  MoveL 3945 to (-46.24, -29.98, -6) mm, rotated rx -180 ry 0 rz 90 deg; joints [72.382, -18.215, 87.048, 0, 21.167, 72.382]
  MoveL 3946 to (-46.24, -29.98, -3) mm, rotated rx 180 ry 0 rz 90 deg; joints [72.382, -18.371, 87.15, 0, 21.221, 72.382]
  Establecer velocidad (1000.0 mm/s)
  MoveL 3947 to (-46.24, -29.98, 10) mm, rotated rx -180 ry 0 rz 90 deg; joints [72.382, -19.042, 87.583, 0, 21.46, 72.382]
  Establecer velocidad (66.7 mm/s)
  MoveL 3948 to (17.19, -67.01, 10) mm, rotated rx 180 ry 0 rz 90 deg; joints [71.851, -17.649, 82.287, 0, 25.361, 71.851]
  MoveL 3949 to (17.19, -67.01, -2.75) mm, rotated rx -180 ry 0 rz 90 deg; joints [71.851, -17.004, 81.861, 0, 25.143, 71.851]
  MoveL 3950 to (17.02, -68.52, -3.16) mm, rotated rx 180 ry 0 rz 90 deg; joints [71.803, -16.977, 81.823, 0, 25.153, 71.803]
  MoveL 3951 to (17.22, -70.03, -3.56) mm, rotated rx 180 ry 0 rz 90 deg; joints [71.757, -16.942, 81.759, 0, 25.183, 71.757]
  MoveL 3952 to (17.75, -71.45, -3.97) mm, rotated rx -180 ry 0 rz 90 deg; joints [71.718, -16.902, 81.673, 0, 25.228, 71.718]
  MoveL 3953 to (18.58, -72.72, -4.37) mm, rotated rx 180 ry 0 rz 90 deg; joints [71.687, -16.856, 81.569, 0, 25.287, 71.687]
  MoveL 3954 to (19.67, -73.78, -4.78) mm, rotated rx 180 ry 0 rz 90 deg; joints [71.665, -16.806, 81.451, 0, 25.356, 71.665]
  MoveL 3955 to (20.97, -74.57, -5.19) mm, rotated rx 180 ry 0 rz 90 deg; joints [71.654, -16.754, 81.324, 0, 25.431, 71.654]
  MoveL 3956 to (22.42, -75.05, -5.59) mm, rotated rx -180 ry 0 rz 90 deg; joints [71.654, -16.701, 81.194, 0, 25.508, 71.654]
  MoveL 3957 to (23.93, -75.17, -6) mm, rotated rx -180 ry 0 rz 90 deg; joints [71.666, -16.649, 81.067, 0, 25.582, 71.666]
  MoveL 3958 to (43.12, -74.95, -6) mm, rotated rx -180 ry 0 rz 90 deg; joints [71.869, -16.251, 79.664, 0, 26.587, 71.869]
  MoveL 3959 to (50.7, -74.82, -6) mm, rotated rx 180 ry 0 rz 90 deg; joints [71.949, -16.089, 79.105, 0, 26.984, 71.949]
  MoveC 3960 to (53.51, -71.7, -6) mm, rotated rx 180 ry 0 rz 90 deg; joints [72.073, -16.05, 78.971, 0, 27.079, 72.073] to (53.65, -67.5, -6) mm, rotated rx 180 ry 0 rz 90 deg; joints [72.203, -16.076, 79.061, 0, 27.015, 72.203]
  MoveL 3961 to (53.54, -67.37, -6) mm, rotated rx -180 ry 0 rz 90 deg; joints [72.206, -16.08, 79.072, 0, 27.007, 72.206]
  MoveL 3962 to (28.6, -38.38, -6) mm, rotated rx -180 ry 0 rz 90 deg; joints [72.864, -16.793, 81.584, 0, 25.21, 72.864]
  MoveL 3963 to (26.1, -35.54, -6) mm, rotated rx 180 ry 0 rz 90 deg; joints [72.929, -16.861, 81.829, 0, 25.032, 72.929]
  MoveL 3964 to (11.85, -24.12, -6) mm, rotated rx 180 ry 0 rz 90 deg; joints [73.154, -17.209, 83.109, 0, 24.1, 73.154]
  MoveC 3965 to (10.01, -23.4, -6) mm, rotated rx 180 ry 0 rz 90 deg; joints [73.159, -17.248, 83.256, 0, 23.993, 73.159] to (8.05, -23.61, -6) mm, rotated rx 180 ry 0 rz 90 deg; joints [73.133, -17.284, 83.391, 0, 23.893, 73.133]
  MoveL 3966 to (7.26, -23.95, -6) mm, rotated rx 180 ry 0 rz 90 deg; joints [73.115, -17.297, 83.44, 0, 23.857, 73.115]
  MoveC 3967 to (6.07, -24.83, -6) mm, rotated rx 180 ry 0 rz 90 deg; joints [73.075, -17.315, 83.507, 0, 23.808, 73.075] to (5.36, -26.14, -6) mm, rotated rx -180 ry 0 rz 90 deg; joints [73.026, -17.321, 83.528, 0, 23.792, 73.026]
  MoveL 3968 to (5.21, -26.67, -6) mm, rotated rx -180 ry 0 rz 90 deg; joints [73.008, -17.321, 83.528, 0, 23.793, 73.008]
  MoveL 3969 to (-6.22, -69.65, -6) mm, rotated rx -180 ry 0 rz 90 deg; joints [71.524, -17.277, 83.363, 0, 23.914, 71.524]
  MoveL 3970 to (-6.48, -70.6, -6) mm, rotated rx 180 ry 0 rz 90 deg; joints [71.492, -17.276, 83.359, 0, 23.917, 71.492]
  MoveC 3971 to (-5.7, -73.8, -6) mm, rotated rx -180 ry 0 rz 90 deg; joints [71.399, -17.241, 83.227, 0, 24.013, 71.399] to (-2.85, -75.47, -6) mm, rotated rx 180 ry 0 rz 90 deg; joints [71.376, -17.176, 82.985, 0, 24.19, 71.376]
  MoveL 3972 to (-2.37, -75.48, -6) mm, rotated rx 180 ry 0 rz 90 deg; joints [71.381, -17.167, 82.951, 0, 24.215, 71.381]
  MoveL 3973 to (23.93, -75.17, -6) mm, rotated rx -180 ry 0 rz 90 deg; joints [71.666, -16.649, 81.067, 0, 25.582, 71.666]
  MoveL 3974 to (23.84, -67.62, -6) mm, rotated rx -180 ry 0 rz 90 deg; joints [71.9, -16.702, 81.254, 0, 25.447, 71.9]
  MoveL 3975 to (23.84, -67.62, -3) mm, rotated rx 180 ry 0 rz 90 deg; joints [71.9, -16.853, 81.356, 0, 25.497, 71.9]
  Establecer velocidad (1000.0 mm/s)
  MoveL 3976 to (23.84, -67.62, 10) mm, rotated rx 180 ry 0 rz 90 deg; joints [71.9, -17.51, 81.791, 0, 25.718, 71.9]
  Establecer velocidad (66.7 mm/s)
  MoveL 3977 to (65.32, -31.32, 10) mm, rotated rx -180 ry 0 rz 90 deg; joints [73.432, -16.868, 79.565, 0, 27.303, 73.432]
  MoveL 3978 to (65.32, -31.32, -2.75) mm, rotated rx 180 ry 0 rz 90 deg; joints [73.432, -16.229, 79.136, 0, 27.093, 73.432]
  MoveL 3979 to (66.82, -31.5, -3.16) mm, rotated rx -180 ry 0 rz 90 deg; joints [73.44, -16.174, 79.005, 0, 27.17, 73.44]
  MoveL 3980 to (68.33, -31.32, -3.56) mm, rotated rx -180 ry 0 rz 90 deg; joints [73.459, -16.122, 78.881, 0, 27.24, 73.459]
  MoveL 3981 to (69.76, -30.81, -3.97) mm, rotated rx 180 ry 0 rz 90 deg; joints [73.488, -16.073, 78.771, 0, 27.302, 73.488]
  MoveL 3982 to (71.04, -29.99, -4.37) mm, rotated rx 180 ry 0 rz 90 deg; joints [73.525, -16.03, 78.679, 0, 27.351, 73.525]
  MoveL 3983 to (72.11, -28.92, -4.78) mm, rotated rx 180 ry 0 rz 90 deg; joints [73.568, -15.993, 78.608, 0, 27.385, 73.568]
  MoveL 3984 to (72.92, -27.63, -5.19) mm, rotated rx 180 ry 0 rz 90 deg; joints [73.615, -15.963, 78.562, 0, 27.401, 73.615]
  MoveL 3985 to (73.42, -26.19, -5.59) mm, rotated rx -180 ry 0 rz 90 deg; joints [73.664, -15.941, 78.542, 0, 27.399, 73.664]
  MoveL 3986 to (73.56, -24.68, -6) mm, rotated rx -180 ry 0 rz 90 deg; joints [73.712, -15.927, 78.551, 0, 27.376, 73.712]
  MoveL 3987 to (73.56, -10.28, -6) mm, rotated rx 180 ry 0 rz 90 deg; joints [74.158, -16.019, 78.865, 0, 27.154, 74.158]
  MoveC 3988 to (71.61, -7.6, -6) mm, rotated rx -180 ry 0 rz 90 deg; joints [74.224, -16.079, 79.069, 0, 27.01, 74.224] to (68.7, -6.02, -6) mm, rotated rx 180 ry 0 rz 90 deg; joints [74.248, -16.152, 79.322, 0, 26.83, 74.248]
  MoveC 3989 to (67.33, -5.86, -6) mm, rotated rx 180 ry 0 rz 90 deg; joints [74.241, -16.183, 79.429, 0, 26.754, 74.241] to (65.97, -6.14, -6) mm, rotated rx 180 ry 0 rz 90 deg; joints [74.22, -16.211, 79.525, 0, 26.686, 74.22]
  MoveL 3990 to (64.91, -7.57, -6) mm, rotated rx -180 ry 0 rz 90 deg; joints [74.166, -16.225, 79.574, 0, 26.651, 74.166]
  MoveL 3991 to (54.87, -21.32, -6) mm, rotated rx -180 ry 0 rz 90 deg; joints [73.646, -16.355, 80.028, 0, 26.327, 73.646]
  MoveL 3992 to (53.21, -23.57, -6) mm, rotated rx -180 ry 0 rz 90 deg; joints [73.561, -16.376, 80.102, 0, 26.275, 73.561]
  MoveC 3993 to (52.43, -26.14, -6) mm, rotated rx 180 ry 0 rz 90 deg; joints [73.474, -16.377, 80.103, 0, 26.274, 73.474] to (53.45, -28.63, -6) mm, rotated rx 180 ry 0 rz 90 deg; joints [73.406, -16.34, 79.973, 0, 26.367, 73.406]
  MoveL 3994 to (66.39, -43.19, -6) mm, rotated rx 180 ry 0 rz 90 deg; joints [73.075, -15.964, 78.676, 0, 27.288, 73.075]
  MoveC 3995 to (68.56, -43.36, -6) mm, rotated rx 180 ry 0 rz 90 deg; joints [73.09, -15.915, 78.508, 0, 27.407, 73.09] to (70.6, -42.58, -6) mm, rotated rx 180 ry 0 rz 90 deg; joints [73.133, -15.875, 78.372, 0, 27.503, 73.133]
  MoveL 3996 to (71.01, -42.29, -6) mm, rotated rx -180 ry 0 rz 90 deg; joints [73.146, -15.867, 78.348, 0, 27.52, 73.146]
  MoveC 3997 to (72.52, -40.87, -6) mm, rotated rx 180 ry 0 rz 90 deg; joints [73.203, -15.843, 78.266, 0, 27.577, 73.203] to (73.56, -39.08, -6) mm, rotated rx -180 ry 0 rz 90 deg; joints [73.268, -15.832, 78.228, 0, 27.604, 73.268]
  MoveL 3998 to (73.56, -24.68, -6) mm, rotated rx -180 ry 0 rz 90 deg; joints [73.712, -15.927, 78.551, 0, 27.376, 73.712]
  MoveL 3999 to (66.01, -24.68, -6) mm, rotated rx 180 ry 0 rz 90 deg; joints [73.644, -16.094, 79.121, 0, 26.973, 73.644]
  MoveL 4000 to (66.01, -24.68, -3) mm, rotated rx 180 ry 0 rz 90 deg; joints [73.644, -16.244, 79.223, 0, 27.021, 73.644]
  Establecer velocidad (1000.0 mm/s)
  MoveL 4001 to (66.01, -24.68, 10) mm, rotated rx -180 ry 0 rz 90 deg; joints [73.644, -16.896, 79.66, 0, 27.236, 73.644]
  Establecer velocidad (66.7 mm/s)
  MoveL 4002 to (37.19, 22.66, 10) mm, rotated rx 180 ry 0 rz 90 deg; joints [74.878, -17.786, 82.781, 0, 25.005, 74.878]
  MoveL 4003 to (37.19, 22.66, -2.75) mm, rotated rx -180 ry 0 rz 90 deg; joints [74.878, -17.14, 82.354, 0, 24.785, 74.878]
  MoveL 4004 to (37.34, 24.17, -3.16) mm, rotated rx -180 ry 0 rz 90 deg; joints [74.928, -17.124, 82.36, 0, 24.765, 74.928]
  MoveL 4005 to (37.12, 25.67, -3.56) mm, rotated rx 180 ry 0 rz 90 deg; joints [74.974, -17.116, 82.391, 0, 24.725, 74.974]
  MoveL 4006 to (36.57, 27.09, -3.97) mm, rotated rx -180 ry 0 rz 90 deg; joints [75.015, -17.114, 82.445, 0, 24.669, 75.015]
  MoveL 4007 to (35.73, 28.35, -4.37) mm, rotated rx 180 ry 0 rz 90 deg; joints [75.048, -17.117, 82.518, 0, 24.599, 75.048]
  MoveL 4008 to (34.62, 29.4, -4.78) mm, rotated rx 180 ry 0 rz 90 deg; joints [75.072, -17.124, 82.605, 0, 24.519, 75.072]
  MoveL 4009 to (33.31, 30.17, -5.19) mm, rotated rx -180 ry 0 rz 90 deg; joints [75.085, -17.133, 82.701, 0, 24.432, 75.085]
  MoveL 4010 to (31.87, 30.63, -5.59) mm, rotated rx 180 ry 0 rz 90 deg; joints [75.088, -17.143, 82.802, 0, 24.342, 75.088]
  MoveL 4011 to (30.35, 30.74, -6) mm, rotated rx 180 ry 0 rz 90 deg; joints [75.078, -17.153, 82.9, 0, 24.253, 75.078]
  MoveL 4012 to (9, 30.22, -6) mm, rotated rx 180 ry 0 rz 90 deg; joints [74.876, -17.556, 84.425, 0, 23.131, 74.876]
  MoveC 4013 to (5.64, 28.68, -6) mm, rotated rx 180 ry 0 rz 90 deg; joints [74.797, -17.611, 84.634, 0, 22.976, 74.797] to (4.7, 25.11, -6) mm, rotated rx 180 ry 0 rz 90 deg; joints [74.672, -17.61, 84.632, 0, 22.978, 74.672]
  MoveL 4014 to (5.03, 24.17, -6) mm, rotated rx -180 ry 0 rz 90 deg; joints [74.645, -17.599, 84.59, 0, 23.009, 74.645]
  MoveL 4015 to (10.58, 8.87, -6) mm, rotated rx 180 ry 0 rz 90 deg; joints [74.2, -17.417, 83.891, 0, 23.526, 74.2]
  MoveC 4016 to (11.12, 7.86, -6) mm, rotated rx 180 ry 0 rz 90 deg; joints [74.172, -17.401, 83.832, 0, 23.569, 74.172] to (11.92, 7.03, -6) mm, rotated rx 180 ry 0 rz 90 deg; joints [74.153, -17.382, 83.758, 0, 23.624, 74.153]
  MoveL 4017 to (28.28, -5.64, -6) mm, rotated rx 180 ry 0 rz 90 deg; joints [73.897, -16.995, 82.317, 0, 24.678, 73.897]
  MoveC 4018 to (30.24, -6.45, -6) mm, rotated rx -180 ry 0 rz 90 deg; joints [73.889, -16.951, 82.158, 0, 24.794, 73.889] to (32.34, -6.16, -6) mm, rotated rx -180 ry 0 rz 90 deg; joints [73.918, -16.911, 82.011, 0, 24.9, 73.918]
  MoveC 4019 to (33.47, -5.59, -6) mm, rotated rx 180 ry 0 rz 90 deg; joints [73.946, -16.892, 81.941, 0, 24.951, 73.946] to (34.36, -4.69, -6) mm, rotated rx 180 ry 0 rz 90 deg; joints [73.983, -16.879, 81.895, 0, 24.984, 73.983]
  MoveL 4020 to (54.3, 23.22, -6) mm, rotated rx -180 ry 0 rz 90 deg; joints [75.042, -16.63, 80.997, 0, 25.633, 75.042]
  MoveL 4021 to (54.77, 23.88, -6) mm, rotated rx 180 ry 0 rz 90 deg; joints [75.067, -16.624, 80.975, 0, 25.648, 75.067]
  MoveC 4022 to (55.09, 24.53, -6) mm, rotated rx 180 ry 0 rz 90 deg; joints [75.09, -16.621, 80.964, 0, 25.656, 75.09] to (55.2, 25.24, -6) mm, rotated rx 180 ry 0 rz 90 deg; joints [75.114, -16.622, 80.97, 0, 25.652, 75.114]
  MoveL 4023 to (55.21, 25.78, -6) mm, rotated rx 180 ry 0 rz 90 deg; joints [75.131, -16.625, 80.98, 0, 25.645, 75.131]
  MoveC 4024 to (54.27, 29.03, -6) mm, rotated rx 180 ry 0 rz 90 deg; joints [75.226, -16.662, 81.113, 0, 25.549, 75.226] to (51.7, 31.24, -6) mm, rotated rx -180 ry 0 rz 90 deg; joints [75.275, -16.727, 81.346, 0, 25.381, 75.275]
  MoveL 4025 to (49.75, 31.21, -6) mm, rotated rx 180 ry 0 rz 90 deg; joints [75.258, -16.767, 81.49, 0, 25.277, 75.258]
  MoveL 4026 to (30.35, 30.74, -6) mm, rotated rx 180 ry 0 rz 90 deg; joints [75.078, -17.153, 82.9, 0, 24.253, 75.078]
  MoveL 4027 to (30.54, 23.19, -6) mm, rotated rx 180 ry 0 rz 90 deg; joints [74.838, -17.109, 82.739, 0, 24.37, 74.838]
  MoveL 4028 to (30.54, 23.19, -3) mm, rotated rx 180 ry 0 rz 90 deg; joints [74.838, -17.262, 82.841, 0, 24.421, 74.838]
  Establecer velocidad (1000.0 mm/s)
  MoveL 4029 to (30.54, 23.19, 10) mm, rotated rx 180 ry 0 rz 90 deg; joints [74.838, -17.922, 83.275, 0, 24.647, 74.838]
  Establecer velocidad (66.7 mm/s)
  MoveL 4030 to (26.5, 66.74, 10) mm, rotated rx 180 ry 0 rz 90 deg; joints [76.21, -18.22, 84.38, 0, 23.84, 76.21]
  MoveL 4031 to (26.5, 66.74, -2.75) mm, rotated rx 180 ry 0 rz 90 deg; joints [76.21, -17.57, 83.955, 0, 23.615, 76.21]
  MoveL 4032 to (26.71, 68.24, -3.16) mm, rotated rx 180 ry 0 rz 90 deg; joints [76.261, -17.553, 83.953, 0, 23.6, 76.261]
  MoveL 4033 to (26.54, 69.75, -3.56) mm, rotated rx 180 ry 0 rz 90 deg; joints [76.309, -17.542, 83.978, 0, 23.564, 76.309]
  MoveL 4034 to (26.05, 71.19, -3.97) mm, rotated rx -180 ry 0 rz 90 deg; joints [76.352, -17.537, 84.025, 0, 23.513, 76.352]
  MoveL 4035 to (25.25, 72.48, -4.37) mm, rotated rx 180 ry 0 rz 90 deg; joints [76.387, -17.538, 84.092, 0, 23.446, 76.387]
  MoveL 4036 to (24.18, 73.57, -4.78) mm, rotated rx 180 ry 0 rz 90 deg; joints [76.414, -17.542, 84.173, 0, 23.369, 76.414]
  MoveL 4037 to (22.9, 74.39, -5.19) mm, rotated rx -180 ry 0 rz 90 deg; joints [76.431, -17.549, 84.266, 0, 23.283, 76.431]
  MoveL 4038 to (21.47, 74.9, -5.59) mm, rotated rx -180 ry 0 rz 90 deg; joints [76.437, -17.558, 84.364, 0, 23.194, 76.437]
  MoveL 4039 to (19.96, 75.06, -6) mm, rotated rx -180 ry 0 rz 90 deg; joints [76.43, -17.566, 84.461, 0, 23.105, 76.43]
  MoveL 4040 to (12.79, 75.15, -6) mm, rotated rx 180 ry 0 rz 90 deg; joints [76.376, -17.698, 84.976, 0, 22.723, 76.376]
  MoveL 4041 to (-28.9, 75.59, -6) mm, rotated rx -180 ry 0 rz 90 deg; joints [76.051, -18.421, 87.908, 0, 20.513, 76.051]
  MoveL 4042 to (-29.63, 75.59, -6) mm, rotated rx -180 ry 0 rz 90 deg; joints [76.045, -18.433, 87.958, 0, 20.475, 76.045]
  MoveC 4043 to (-32.33, 72.16, -6) mm, rotated rx 180 ry 0 rz 90 deg; joints [75.907, -18.463, 88.086, 0, 20.377, 75.907] to (-31.86, 67.82, -6) mm, rotated rx -180 ry 0 rz 90 deg; joints [75.765, -18.438, 87.978, 0, 20.46, 75.765]
  MoveL 4044 to (-10.84, 54.49, -6) mm, rotated rx 180 ry 0 rz 90 deg; joints [75.5, -18.027, 86.281, 0, 21.747, 75.5]
  MoveC 4045 to (-9.04, 53.75, -6) mm, rotated rx 180 ry 0 rz 90 deg; joints [75.491, -17.993, 86.141, 0, 21.852, 75.491] to (-7.11, 53.59, -6) mm, rotated rx -180 ry 0 rz 90 deg; joints [75.502, -17.958, 86.002, 0, 21.956, 75.502]
  MoveL 4046 to (37.91, 56.91, -6) mm, rotated rx -180 ry 0 rz 90 deg; joints [75.984, -17.137, 82.841, 0, 24.296, 75.984]
  MoveC 4047 to (53.8, 58.26, -6) mm, rotated rx -180 ry 0 rz 90 deg; joints [76.153, -16.825, 81.7, 0, 25.126, 76.153] to (69.65, 59.95, -6) mm, rotated rx -180 ry 0 rz 90 deg; joints [76.331, -16.504, 80.551, 0, 25.953, 76.331]
  MoveC 4048 to (71.89, 61.11, -6) mm, rotated rx -180 ry 0 rz 90 deg; joints [76.385, -16.463, 80.405, 0, 26.058, 76.385] to (72.78, 63.46, -6) mm, rotated rx 180 ry 0 rz 90 deg; joints [76.467, -16.456, 80.38, 0, 26.075, 76.467]
  MoveL 4049 to (72.78, 69.65, -6) mm, rotated rx 180 ry 0 rz 90 deg; joints [76.663, -16.487, 80.491, 0, 25.996, 76.663]
  MoveL 4050 to (72.76, 70.26, -6) mm, rotated rx -180 ry 0 rz 90 deg; joints [76.682, -16.491, 80.503, 0, 25.987, 76.682]
  MoveC 4051 to (71.8, 72.55, -6) mm, rotated rx 180 ry 0 rz 90 deg; joints [76.748, -16.523, 80.617, 0, 25.906, 76.748] to (69.53, 73.57, -6) mm, rotated rx -180 ry 0 rz 90 deg; joints [76.763, -16.575, 80.804, 0, 25.771, 76.763]
  MoveC 4052 to (45.44, 74.54, -6) mm, rotated rx 180 ry 0 rz 90 deg; joints [76.612, -17.073, 82.605, 0, 24.468, 76.612] to (21.32, 75.04, -6) mm, rotated rx -180 ry 0 rz 90 deg; joints [76.44, -17.54, 84.363, 0, 23.177, 76.44]
  MoveL 4053 to (19.96, 75.06, -6) mm, rotated rx -180 ry 0 rz 90 deg; joints [76.43, -17.566, 84.461, 0, 23.105, 76.43]
  MoveL 4054 to (19.87, 67.51, -6) mm, rotated rx -180 ry 0 rz 90 deg; joints [76.182, -17.533, 84.336, 0, 23.197, 76.182]
  MoveL 4055 to (19.87, 67.51, -3) mm, rotated rx 180 ry 0 rz 90 deg; joints [76.182, -17.687, 84.437, 0, 23.249, 76.182]
  Establecer velocidad (1000.0 mm/s)
  MoveL 4056 to (19.87, 67.51, 10) mm, rotated rx 180 ry 0 rz 90 deg; joints [76.182, -18.351, 84.871, 0, 23.48, 76.182]
  Establecer velocidad (66.7 mm/s)
  MoveL 4057 to (26.49, 66.5, 10) mm, rotated rx -180 ry 0 rz 90 deg; joints [76.203, -18.219, 84.377, 0, 23.843, 76.203]
  MoveL 4058 to (26.49, 66.5, -3) mm, rotated rx 180 ry 0 rz 90 deg; joints [76.203, -17.557, 83.943, 0, 23.614, 76.203]
  MoveL 4059 to (26.7, 68, -3.41) mm, rotated rx -180 ry 0 rz 90 deg; joints [76.253, -17.539, 83.941, 0, 23.598, 76.253]
  MoveL 4060 to (26.54, 69.51, -3.81) mm, rotated rx -180 ry 0 rz 90 deg; joints [76.301, -17.528, 83.966, 0, 23.563, 76.301]
  MoveL 4061 to (26.04, 70.95, -4.22) mm, rotated rx 180 ry 0 rz 90 deg; joints [76.344, -17.524, 84.013, 0, 23.511, 76.344]
  MoveL 4062 to (25.24, 72.25, -4.63) mm, rotated rx -180 ry 0 rz 90 deg; joints [76.38, -17.524, 84.079, 0, 23.445, 76.38]
  MoveL 4063 to (24.18, 73.33, -5.03) mm, rotated rx -180 ry 0 rz 90 deg; joints [76.407, -17.528, 84.161, 0, 23.367, 76.407]
  MoveL 4064 to (22.9, 74.15, -5.44) mm, rotated rx 180 ry 0 rz 90 deg; joints [76.423, -17.535, 84.254, 0, 23.282, 76.423]
  MoveL 4065 to (21.47, 74.67, -5.84) mm, rotated rx 180 ry 0 rz 90 deg; joints [76.429, -17.544, 84.352, 0, 23.192, 76.429]
  MoveL 4066 to (19.96, 74.83, -6.25) mm, rotated rx -180 ry 0 rz 90 deg; joints [76.422, -17.552, 84.449, 0, 23.103, 76.422]
  MoveL 4067 to (16.58, 74.87, -6.25) mm, rotated rx 180 ry 0 rz 90 deg; joints [76.397, -17.615, 84.692, 0, 22.923, 76.397]
  MoveL 4068 to (-29.04, 75.36, -6.25) mm, rotated rx -180 ry 0 rz 90 deg; joints [76.042, -18.41, 87.905, 0, 20.504, 76.042]
  MoveC 4069 to (-31.69, 71.97, -6.25) mm, rotated rx -180 ry 0 rz 90 deg; joints [75.906, -18.439, 88.029, 0, 20.409, 75.906] to (-31.22, 67.7, -6.25) mm, rotated rx 180 ry 0 rz 90 deg; joints [75.766, -18.414, 87.923, 0, 20.49, 75.766]
  MoveL 4070 to (-10.9, 54.79, -6.25) mm, rotated rx 180 ry 0 rz 90 deg; joints [75.509, -18.017, 86.282, 0, 21.735, 75.509]
  MoveC 4071 to (-9.09, 53.98, -6.25) mm, rotated rx -180 ry 0 rz 90 deg; joints [75.498, -17.982, 86.14, 0, 21.842, 75.498] to (-7.11, 53.8, -6.25) mm, rotated rx -180 ry 0 rz 90 deg; joints [75.509, -17.946, 85.998, 0, 21.949, 75.509]
  MoveL 4072 to (36.88, 57.07, -6.25) mm, rotated rx 180 ry 0 rz 90 deg; joints [75.98, -17.145, 82.911, 0, 24.235, 75.98]
  MoveC 4073 to (53.18, 58.48, -6.25) mm, rotated rx -180 ry 0 rz 90 deg; joints [76.156, -16.826, 81.741, 0, 25.085, 76.156] to (69.44, 60.27, -6.25) mm, rotated rx 180 ry 0 rz 90 deg; joints [76.34, -16.498, 80.564, 0, 25.933, 76.34]
  MoveC 4074 to (71.55, 61.36, -6.25) mm, rotated rx 180 ry 0 rz 90 deg; joints [76.39, -16.458, 80.426, 0, 26.032, 76.39] to (72.45, 63.55, -6.25) mm, rotated rx 180 ry 0 rz 90 deg; joints [76.467, -16.451, 80.398, 0, 26.052, 76.467]
  MoveL 4075 to (72.46, 63.97, -6.25) mm, rotated rx -180 ry 0 rz 90 deg; joints [76.48, -16.452, 80.405, 0, 26.047, 76.48]
  MoveL 4076 to (72.46, 70.25, -6.25) mm, rotated rx -180 ry 0 rz 90 deg; joints [76.68, -16.484, 80.518, 0, 25.967, 76.68]
  MoveL 4077 to (72.45, 70.31, -6.25) mm, rotated rx -180 ry 0 rz 90 deg; joints [76.681, -16.485, 80.519, 0, 25.965, 76.681]
  MoveC 4078 to (71.41, 72.35, -6.25) mm, rotated rx -180 ry 0 rz 90 deg; joints [76.738, -16.517, 80.634, 0, 25.883, 76.738] to (69.3, 73.24, -6.25) mm, rotated rx 180 ry 0 rz 90 deg; joints [76.751, -16.566, 80.807, 0, 25.759, 76.751]
  MoveC 4079 to (45.79, 74.26, -6.25) mm, rotated rx 180 ry 0 rz 90 deg; joints [76.605, -17.052, 82.566, 0, 24.486, 76.605] to (22.27, 74.8, -6.25) mm, rotated rx 180 ry 0 rz 90 deg; joints [76.44, -17.509, 84.282, 0, 23.226, 76.44]
  MoveL 4080 to (19.96, 74.83, -6.25) mm, rotated rx -180 ry 0 rz 90 deg; joints [76.422, -17.552, 84.449, 0, 23.103, 76.422]
  MoveL 4081 to (19.86, 67.28, -6.25) mm, rotated rx 180 ry 0 rz 90 deg; joints [76.175, -17.519, 84.324, 0, 23.196, 76.175]
  MoveL 4082 to (19.86, 67.28, -3.25) mm, rotated rx -180 ry 0 rz 90 deg; joints [76.175, -17.673, 84.425, 0, 23.247, 76.175]
  Establecer velocidad (1000.0 mm/s)
  MoveL 4083 to (19.86, 67.28, 10) mm, rotated rx 180 ry 0 rz 90 deg; joints [76.175, -18.35, 84.867, 0, 23.482, 76.175]
  Establecer velocidad (66.7 mm/s)
  MoveL 4084 to (36.98, 22.41, 10) mm, rotated rx 180 ry 0 rz 90 deg; joints [74.868, -17.788, 82.79, 0, 24.998, 74.868]
  MoveL 4085 to (36.98, 22.41, -3) mm, rotated rx 180 ry 0 rz 90 deg; joints [74.868, -17.13, 82.356, 0, 24.774, 74.868]
  MoveL 4086 to (37.13, 23.92, -3.41) mm, rotated rx 180 ry 0 rz 90 deg; joints [74.918, -17.114, 82.361, 0, 24.753, 74.918]
  MoveL 4087 to (36.92, 25.42, -3.81) mm, rotated rx 180 ry 0 rz 90 deg; joints [74.964, -17.106, 82.393, 0, 24.713, 74.964]
  MoveL 4088 to (36.37, 26.84, -4.22) mm, rotated rx -180 ry 0 rz 90 deg; joints [75.005, -17.104, 82.446, 0, 24.658, 75.005]
  MoveL 4089 to (35.53, 28.1, -4.63) mm, rotated rx -180 ry 0 rz 90 deg; joints [75.038, -17.107, 82.519, 0, 24.588, 75.038]
  MoveL 4090 to (34.42, 29.14, -5.03) mm, rotated rx 180 ry 0 rz 90 deg; joints [75.062, -17.114, 82.606, 0, 24.508, 75.062]
  MoveL 4091 to (33.11, 29.92, -5.44) mm, rotated rx -180 ry 0 rz 90 deg; joints [75.076, -17.123, 82.702, 0, 24.42, 75.076]
  MoveL 4092 to (31.67, 30.38, -5.84) mm, rotated rx 180 ry 0 rz 90 deg; joints [75.078, -17.133, 82.803, 0, 24.33, 75.078]
  MoveL 4093 to (30.15, 30.49, -6.25) mm, rotated rx 180 ry 0 rz 90 deg; joints [75.068, -17.142, 82.901, 0, 24.242, 75.068]
  MoveL 4094 to (9, 29.99, -6.25) mm, rotated rx 180 ry 0 rz 90 deg; joints [74.869, -17.542, 84.412, 0, 23.13, 74.869]
  MoveC 4095 to (5.91, 28.44, -6.25) mm, rotated rx 180 ry 0 rz 90 deg; joints [74.791, -17.592, 84.602, 0, 22.989, 74.791] to (4.97, 25.11, -6.25) mm, rotated rx 180 ry 0 rz 90 deg; joints [74.675, -17.592, 84.604, 0, 22.988, 74.675]
  MoveL 4096 to (5.21, 24.37, -6.25) mm, rotated rx 180 ry 0 rz 90 deg; joints [74.653, -17.584, 84.573, 0, 23.011, 74.653]
  MoveL 4097 to (10.79, 9, -6.25) mm, rotated rx 180 ry 0 rz 90 deg; joints [74.206, -17.401, 83.87, 0, 23.531, 74.206]
  MoveC 4098 to (11.37, 7.95, -6.25) mm, rotated rx 180 ry 0 rz 90 deg; joints [74.177, -17.384, 83.808, 0, 23.576, 74.177] to (12.21, 7.11, -6.25) mm, rotated rx -180 ry 0 rz 90 deg; joints [74.158, -17.364, 83.73, 0, 23.634, 74.158]
  MoveL 4099 to (27.96, -5.07, -6.25) mm, rotated rx -180 ry 0 rz 90 deg; joints [73.912, -16.992, 82.344, 0, 24.648, 73.912]
  MoveL 4100 to (28.9, -5.75, -6.25) mm, rotated rx -180 ry 0 rz 90 deg; joints [73.899, -16.969, 82.261, 0, 24.708, 73.899]
  MoveC 4101 to (30.3, -6.12, -6.25) mm, rotated rx -180 ry 0 rz 90 deg; joints [73.9, -16.939, 82.152, 0, 24.787, 73.9] to (31.75, -6.02, -6.25) mm, rotated rx -180 ry 0 rz 90 deg; joints [73.916, -16.911, 82.049, 0, 24.862, 73.916]
  MoveC 4102 to (33.22, -5.39, -6.25) mm, rotated rx -180 ry 0 rz 90 deg; joints [73.95, -16.885, 81.955, 0, 24.93, 73.95] to (34.37, -4.27, -6.25) mm, rotated rx -180 ry 0 rz 90 deg; joints [73.996, -16.869, 81.894, 0, 24.974, 73.996]
  MoveL 4103 to (52.64, 21.32, -6.25) mm, rotated rx -180 ry 0 rz 90 deg; joints [74.968, -16.641, 81.073, 0, 25.567, 74.968]
  MoveL 4104 to (54.49, 23.94, -6.25) mm, rotated rx 180 ry 0 rz 90 deg; joints [75.067, -16.617, 80.989, 0, 25.628, 75.067]
  MoveC 4105 to (54.19, 28.03, -6.25) mm, rotated rx 180 ry 0 rz 90 deg; joints [75.194, -16.646, 81.091, 0, 25.554, 75.194] to (51.31, 30.95, -6.25) mm, rotated rx 180 ry 0 rz 90 deg; joints [75.262, -16.721, 81.362, 0, 25.36, 75.262]
  MoveL 4106 to (47.86, 30.9, -6.25) mm, rotated rx -180 ry 0 rz 90 deg; joints [75.232, -16.791, 81.615, 0, 25.176, 75.232]
  MoveL 4107 to (30.15, 30.49, -6.25) mm, rotated rx 180 ry 0 rz 90 deg; joints [75.068, -17.142, 82.901, 0, 24.242, 75.068]
  MoveL 4108 to (30.33, 22.94, -6.25) mm, rotated rx -180 ry 0 rz 90 deg; joints [74.828, -17.099, 82.74, 0, 24.359, 74.828]
  MoveL 4109 to (30.33, 22.94, -3.25) mm, rotated rx 180 ry 0 rz 90 deg; joints [74.828, -17.252, 82.842, 0, 24.41, 74.828]
  Establecer velocidad (1000.0 mm/s)
  MoveL 4110 to (30.33, 22.94, 10) mm, rotated rx 180 ry 0 rz 90 deg; joints [74.828, -17.924, 83.285, 0, 24.64, 74.828]
  Establecer velocidad (66.7 mm/s)
  MoveL 4111 to (65.05, -31.33, 10) mm, rotated rx 180 ry 0 rz 90 deg; joints [73.429, -16.874, 79.585, 0, 27.289, 73.429]
  MoveL 4112 to (65.05, -31.33, -3) mm, rotated rx -180 ry 0 rz 90 deg; joints [73.429, -16.222, 79.148, 0, 27.075, 73.429]
  MoveL 4113 to (66.55, -31.52, -3.41) mm, rotated rx 180 ry 0 rz 90 deg; joints [73.437, -16.168, 79.017, 0, 27.151, 73.437]
  MoveL 4114 to (68.06, -31.33, -3.81) mm, rotated rx 180 ry 0 rz 90 deg; joints [73.456, -16.115, 78.893, 0, 27.222, 73.456]
  MoveL 4115 to (69.49, -30.82, -4.22) mm, rotated rx -180 ry 0 rz 90 deg; joints [73.485, -16.067, 78.783, 0, 27.284, 73.485]
  MoveL 4116 to (70.77, -30.01, -4.63) mm, rotated rx 180 ry 0 rz 90 deg; joints [73.522, -16.023, 78.691, 0, 27.333, 73.522]
  MoveL 4117 to (71.84, -28.93, -5.03) mm, rotated rx -180 ry 0 rz 90 deg; joints [73.565, -15.986, 78.62, 0, 27.366, 73.565]
  MoveL 4118 to (72.65, -27.64, -5.44) mm, rotated rx -180 ry 0 rz 90 deg; joints [73.613, -15.957, 78.574, 0, 27.383, 73.613]
  MoveL 4119 to (73.15, -26.2, -5.84) mm, rotated rx -180 ry 0 rz 90 deg; joints [73.661, -15.934, 78.554, 0, 27.38, 73.661]
  MoveL 4120 to (73.28, -24.69, -6.25) mm, rotated rx -180 ry 0 rz 90 deg; joints [73.709, -15.921, 78.563, 0, 27.358, 73.709]
  MoveL 4121 to (73.28, -11, -6.25) mm, rotated rx -180 ry 0 rz 90 deg; joints [74.133, -16.008, 78.862, 0, 27.147, 74.133]
  MoveC 4122 to (71.09, -8.09, -6.25) mm, rotated rx 180 ry 0 rz 90 deg; joints [74.204, -16.075, 79.09, 0, 26.985, 74.204] to (67.76, -6.62, -6.25) mm, rotated rx 180 ry 0 rz 90 deg; joints [74.221, -16.156, 79.372, 0, 26.785, 74.221]
  MoveC 4123 to (66.71, -6.6, -6.25) mm, rotated rx 180 ry 0 rz 90 deg; joints [74.212, -16.179, 79.451, 0, 26.728, 74.212] to (65.72, -6.94, -6.25) mm, rotated rx 180 ry 0 rz 90 deg; joints [74.193, -16.199, 79.518, 0, 26.681, 74.193]
  MoveL 4124 to (53.8, -23.22, -6.25) mm, rotated rx -180 ry 0 rz 90 deg; joints [73.578, -16.353, 80.057, 0, 26.296, 73.578]
  MoveL 4125 to (53.37, -23.87, -6.25) mm, rotated rx -180 ry 0 rz 90 deg; joints [73.553, -16.358, 80.075, 0, 26.284, 73.553]
  MoveC 4126 to (52.75, -26.09, -6.25) mm, rotated rx -180 ry 0 rz 90 deg; joints [73.478, -16.358, 80.072, 0, 26.286, 73.478] to (53.54, -28.26, -6.25) mm, rotated rx -180 ry 0 rz 90 deg; joints [73.418, -16.327, 79.965, 0, 26.362, 73.418]
  MoveL 4127 to (54.9, -29.85, -6.25) mm, rotated rx 180 ry 0 rz 90 deg; joints [73.381, -16.288, 79.829, 0, 26.459, 73.381]
  MoveL 4128 to (66.21, -42.58, -6.25) mm, rotated rx -180 ry 0 rz 90 deg; joints [73.092, -15.959, 78.695, 0, 27.265, 73.092]
  MoveC 4129 to (68.5, -42.7, -6.25) mm, rotated rx 180 ry 0 rz 90 deg; joints [73.11, -15.908, 78.52, 0, 27.388, 73.11] to (70.6, -41.79, -6.25) mm, rotated rx 180 ry 0 rz 90 deg; joints [73.157, -15.867, 78.381, 0, 27.486, 73.157]
  MoveL 4130 to (71.12, -41.39, -6.25) mm, rotated rx 180 ry 0 rz 90 deg; joints [73.175, -15.859, 78.351, 0, 27.507, 73.175]
  MoveC 4131 to (72.42, -40.04, -6.25) mm, rotated rx 180 ry 0 rz 90 deg; joints [73.228, -15.839, 78.284, 0, 27.555, 73.228] to (73.28, -38.38, -6.25) mm, rotated rx 180 ry 0 rz 90 deg; joints [73.287, -15.83, 78.256, 0, 27.574, 73.287]
  MoveL 4132 to (73.28, -24.69, -6.25) mm, rotated rx -180 ry 0 rz 90 deg; joints [73.709, -15.921, 78.563, 0, 27.358, 73.709]
  MoveL 4133 to (65.74, -24.69, -6.25) mm, rotated rx 180 ry 0 rz 90 deg; joints [73.641, -16.087, 79.132, 0, 26.955, 73.641]
  MoveL 4134 to (65.74, -24.69, -3.25) mm, rotated rx -180 ry 0 rz 90 deg; joints [73.641, -16.238, 79.235, 0, 27.003, 73.641]
  Establecer velocidad (1000.0 mm/s)
  MoveL 4135 to (65.74, -24.69, 10) mm, rotated rx 180 ry 0 rz 90 deg; joints [73.641, -16.902, 79.681, 0, 27.221, 73.641]
  Establecer velocidad (66.7 mm/s)
  MoveL 4136 to (17.44, -66.81, 10) mm, rotated rx 180 ry 0 rz 90 deg; joints [71.86, -17.645, 82.274, 0, 25.371, 71.86]
  MoveL 4137 to (17.44, -66.81, -3) mm, rotated rx -180 ry 0 rz 90 deg; joints [71.86, -16.988, 81.839, 0, 25.149, 71.86]
  MoveL 4138 to (17.27, -68.32, -3.41) mm, rotated rx 180 ry 0 rz 90 deg; joints [71.811, -16.96, 81.801, 0, 25.159, 71.811]
  MoveL 4139 to (17.48, -69.82, -3.81) mm, rotated rx 180 ry 0 rz 90 deg; joints [71.766, -16.926, 81.737, 0, 25.189, 71.766]
  MoveL 4140 to (18.01, -71.25, -4.22) mm, rotated rx 180 ry 0 rz 90 deg; joints [71.727, -16.885, 81.651, 0, 25.234, 71.727]
  MoveL 4141 to (18.84, -72.52, -4.63) mm, rotated rx 180 ry 0 rz 90 deg; joints [71.696, -16.84, 81.547, 0, 25.293, 71.696]
  MoveL 4142 to (19.93, -73.57, -5.03) mm, rotated rx -180 ry 0 rz 90 deg; joints [71.675, -16.79, 81.429, 0, 25.361, 71.675]
  MoveL 4143 to (21.23, -74.36, -5.44) mm, rotated rx 180 ry 0 rz 90 deg; joints [71.663, -16.738, 81.302, 0, 25.436, 71.663]
  MoveL 4144 to (22.67, -74.84, -5.84) mm, rotated rx 180 ry 0 rz 90 deg; joints [71.663, -16.685, 81.171, 0, 25.513, 71.663]
  MoveL 4145 to (24.19, -74.96, -6.25) mm, rotated rx -180 ry 0 rz 90 deg; joints [71.675, -16.633, 81.045, 0, 25.588, 71.675]
  MoveC 4146 to (36.97, -74.78, -6.25) mm, rotated rx -180 ry 0 rz 90 deg; joints [71.812, -16.37, 80.114, 0, 26.256, 71.812] to (49.75, -74.58, -6.25) mm, rotated rx 180 ry 0 rz 90 deg; joints [71.947, -16.099, 79.173, 0, 26.926, 71.947]
  MoveL 4147 to (50.59, -74.39, -6.25) mm, rotated rx 180 ry 0 rz 90 deg; joints [71.961, -16.082, 79.115, 0, 26.967, 71.961]
  MoveL 4148 to (50.7, -74.32, -6.25) mm, rotated rx 180 ry 0 rz 90 deg; joints [71.964, -16.08, 79.108, 0, 26.972, 71.964]
  MoveC 4149 to (53.08, -71.2, -6.25) mm, rotated rx -180 ry 0 rz 90 deg; joints [72.084, -16.05, 79.006, 0, 27.044, 72.084] to (53.13, -67.28, -6.25) mm, rotated rx 180 ry 0 rz 90 deg; joints [72.205, -16.077, 79.097, 0, 26.98, 72.205]
  MoveL 4150 to (50.7, -64.44, -6.25) mm, rotated rx 180 ry 0 rz 90 deg; joints [72.269, -16.149, 79.346, 0, 26.803, 72.269]
  MoveL 4151 to (26.66, -36.48, -6.25) mm, rotated rx -180 ry 0 rz 90 deg; joints [72.905, -16.831, 81.758, 0, 25.073, 72.905]
  MoveL 4152 to (26.06, -35.81, -6.25) mm, rotated rx 180 ry 0 rz 90 deg; joints [72.92, -16.847, 81.817, 0, 25.03, 72.92]
  MoveL 4153 to (25.76, -35.54, -6.25) mm, rotated rx -180 ry 0 rz 90 deg; joints [72.926, -16.855, 81.845, 0, 25.01, 72.926]
  MoveL 4154 to (11.74, -24.32, -6.25) mm, rotated rx -180 ry 0 rz 90 deg; joints [73.146, -17.197, 83.103, 0, 24.093, 73.146]
  MoveC 4155 to (8.32, -23.9, -6.25) mm, rotated rx 180 ry 0 rz 90 deg; joints [73.127, -17.265, 83.357, 0, 23.907, 73.127] to (5.63, -26.06, -6.25) mm, rotated rx 180 ry 0 rz 90 deg; joints [73.031, -17.303, 83.502, 0, 23.801, 73.031]
  MoveL 4156 to (5.36, -27.01, -6.25) mm, rotated rx 180 ry 0 rz 90 deg; joints [72.998, -17.303, 83.501, 0, 23.802, 72.998]
  MoveL 4157 to (-6.24, -70.6, -6.25) mm, rotated rx -180 ry 0 rz 90 deg; joints [71.494, -17.258, 83.333, 0, 23.925, 71.494]
  MoveC 4158 to (-5.31, -73.76, -6.25) mm, rotated rx 180 ry 0 rz 90 deg; joints [71.404, -17.221, 83.192, 0, 24.028, 71.404] to (-2.37, -75.25, -6.25) mm, rotated rx 180 ry 0 rz 90 deg; joints [71.388, -17.155, 82.948, 0, 24.207, 71.388]
  MoveC 4159 to (10.91, -75.12, -6.25) mm, rotated rx -180 ry 0 rz 90 deg; joints [71.532, -16.898, 82.002, 0, 24.897, 71.532] to (24.19, -74.96, -6.25) mm, rotated rx -180 ry 0 rz 90 deg; joints [71.675, -16.633, 81.045, 0, 25.588, 71.675]
  MoveL 4160 to (24.09, -67.41, -6.25) mm, rotated rx 180 ry 0 rz 90 deg; joints [71.909, -16.685, 81.233, 0, 25.453, 71.909]
  MoveL 4161 to (24.09, -67.41, -3.25) mm, rotated rx 180 ry 0 rz 90 deg; joints [71.909, -16.837, 81.334, 0, 25.502, 71.909]
  Establecer velocidad (1000.0 mm/s)
  MoveL 4162 to (24.09, -67.41, 10) mm, rotated rx 180 ry 0 rz 90 deg; joints [71.909, -17.506, 81.778, 0, 25.728, 71.909]
  Establecer velocidad (66.7 mm/s)
  MoveL 4163 to (-34.29, -51.62, 10) mm, rotated rx 180 ry 0 rz 90 deg; joints [71.804, -18.716, 86.28, 0, 22.436, 71.804]
  MoveL 4164 to (-34.29, -51.62, -3) mm, rotated rx -180 ry 0 rz 90 deg; joints [71.804, -18.048, 85.847, 0, 22.201, 71.804]
  MoveL 4165 to (-32.88, -52.17, -3.41) mm, rotated rx 180 ry 0 rz 90 deg; joints [71.801, -17.999, 85.723, 0, 22.277, 71.801]
  MoveL 4166 to (-31.37, -52.38, -3.81) mm, rotated rx 180 ry 0 rz 90 deg; joints [71.81, -17.951, 85.6, 0, 22.351, 71.81]
  MoveL 4167 to (-29.86, -52.24, -4.22) mm, rotated rx -180 ry 0 rz 90 deg; joints [71.83, -17.904, 85.485, 0, 22.42, 71.83]
  MoveL 4168 to (-28.41, -51.78, -4.63) mm, rotated rx -180 ry 0 rz 90 deg; joints [71.861, -17.861, 85.381, 0, 22.479, 71.861]
  MoveL 4169 to (-27.1, -51, -5.03) mm, rotated rx -180 ry 0 rz 90 deg; joints [71.899, -17.821, 85.294, 0, 22.527, 71.899]
  MoveL 4170 to (-26, -49.96, -5.44) mm, rotated rx 180 ry 0 rz 90 deg; joints [71.945, -17.787, 85.227, 0, 22.559, 71.945]
  MoveL 4171 to (-25.16, -48.69, -5.84) mm, rotated rx -180 ry 0 rz 90 deg; joints [71.994, -17.758, 85.184, 0, 22.575, 71.994]
  MoveL 4172 to (-24.64, -47.27, -6.25) mm, rotated rx 180 ry 0 rz 90 deg; joints [72.046, -17.736, 85.166, 0, 22.57, 72.046]
  MoveL 4173 to (-18.29, -22.89, -6.25) mm, rotated rx 180 ry 0 rz 90 deg; joints [72.898, -17.76, 85.261, 0, 22.5, 72.898]
  MoveC 4174 to (-18.85, -19.41, -6.25) mm, rotated rx 180 ry 0 rz 90 deg; joints [73.005, -17.789, 85.374, 0, 22.415, 73.005] to (-21.8, -17.48, -6.25) mm, rotated rx -180 ry 0 rz 90 deg; joints [73.038, -17.852, 85.621, 0, 22.231, 73.038]
  MoveC 4175 to (-22.65, -17.51, -6.25) mm, rotated rx 180 ry 0 rz 90 deg; joints [73.029, -17.866, 85.68, 0, 22.187, 73.029] to (-23.49, -17.63, -6.25) mm, rotated rx -180 ry 0 rz 90 deg; joints [73.016, -17.881, 85.736, 0, 22.145, 73.016]
  MoveL 4176 to (-72.48, -28.06, -6.25) mm, rotated rx -180 ry 0 rz 90 deg; joints [72.169, -18.631, 88.858, 0, 19.774, 72.169]
  MoveC 4177 to (-74.99, -29.6, -6.25) mm, rotated rx -180 ry 0 rz 90 deg; joints [72.09, -18.662, 88.992, 0, 19.67, 72.09] to (-75.97, -32.38, -6.25) mm, rotated rx 180 ry 0 rz 90 deg; joints [71.988, -18.663, 88.998, 0, 19.665, 71.988]
  MoveL 4178 to (-75.97, -71.05, -6.25) mm, rotated rx -180 ry 0 rz 90 deg; joints [70.711, -18.461, 88.125, 0, 20.337, 70.711]
  MoveC 4179 to (-75.13, -73.56, -6.25) mm, rotated rx 180 ry 0 rz 90 deg; joints [70.639, -18.434, 88.01, 0, 20.424, 70.639] to (-72.96, -75.06, -6.25) mm, rotated rx -180 ry 0 rz 90 deg; joints [70.615, -18.391, 87.828, 0, 20.563, 70.615]
  MoveC 4180 to (-72.02, -75.26, -6.25) mm, rotated rx -180 ry 0 rz 90 deg; joints [70.619, -18.375, 87.76, 0, 20.615, 70.619] to (-71.06, -75.33, -6.25) mm, rotated rx 180 ry 0 rz 90 deg; joints [70.628, -18.36, 87.694, 0, 20.665, 70.628]
  MoveL 4181 to (-35.36, -75.05, -6.25) mm, rotated rx -180 ry 0 rz 90 deg; joints [71.038, -17.762, 85.266, 0, 22.496, 71.038]
  MoveC 4182 to (-32.59, -74.09, -6.25) mm, rotated rx -180 ry 0 rz 90 deg; joints [71.099, -17.719, 85.098, 0, 22.621, 71.099] to (-30.99, -71.65, -6.25) mm, rotated rx 180 ry 0 rz 90 deg; joints [71.195, -17.705, 85.044, 0, 22.661, 71.195]
  MoveL 4183 to (-24.64, -47.27, -6.25) mm, rotated rx 180 ry 0 rz 90 deg; joints [72.046, -17.736, 85.166, 0, 22.57, 72.046]
  MoveL 4184 to (-31.95, -45.36, -6.25) mm, rotated rx -180 ry 0 rz 90 deg; joints [72.031, -17.876, 85.716, 0, 22.159, 72.031]
  MoveL 4185 to (-31.95, -45.36, -3.25) mm, rotated rx 180 ry 0 rz 90 deg; joints [72.031, -18.03, 85.818, 0, 22.212, 72.031]
  Establecer velocidad (1000.0 mm/s)
  MoveL 4186 to (-31.95, -45.36, 10) mm, rotated rx 180 ry 0 rz 90 deg; joints [72.031, -18.711, 86.259, 0, 22.451, 72.031]
  Establecer velocidad (66.7 mm/s)
  MoveL 4187 to (-67.73, 36.21, 10) mm, rotated rx -180 ry 0 rz 90 deg; joints [74.375, -19.702, 90.378, 0, 19.324, 74.375]
  MoveL 4188 to (-67.73, 36.21, -3) mm, rotated rx -180 ry 0 rz 90 deg; joints [74.375, -19.022, 89.945, 0, 19.077, 74.375]
  MoveL 4189 to (-69.24, 36.39, -3.41) mm, rotated rx -180 ry 0 rz 90 deg; joints [74.367, -19.024, 90.036, 0, 18.988, 74.367]
  MoveL 4190 to (-70.74, 36.21, -3.81) mm, rotated rx 180 ry 0 rz 90 deg; joints [74.346, -19.024, 90.12, 0, 18.905, 74.346]
  MoveL 4191 to (-72.17, 35.7, -4.22) mm, rotated rx -180 ry 0 rz 90 deg; joints [74.315, -19.022, 90.192, 0, 18.83, 74.315]
  MoveL 4192 to (-73.46, 34.88, -4.63) mm, rotated rx 180 ry 0 rz 90 deg; joints [74.275, -19.016, 90.249, 0, 18.767, 74.275]
  MoveL 4193 to (-74.53, 33.8, -5.03) mm, rotated rx 180 ry 0 rz 90 deg; joints [74.228, -19.006, 90.286, 0, 18.72, 74.228]
  MoveL 4194 to (-75.33, 32.51, -5.44) mm, rotated rx -180 ry 0 rz 90 deg; joints [74.177, -18.991, 90.302, 0, 18.689, 74.177]
  MoveL 4195 to (-75.83, 31.08, -5.84) mm, rotated rx 180 ry 0 rz 90 deg; joints [74.123, -18.971, 90.294, 0, 18.677, 74.123]
  MoveL 4196 to (-75.97, 29.57, -6.25) mm, rotated rx 180 ry 0 rz 90 deg; joints [74.07, -18.945, 90.261, 0, 18.685, 74.07]
  MoveL 4197 to (-75.97, 1.42, -6.25) mm, rotated rx -180 ry 0 rz 90 deg; joints [73.118, -18.823, 89.708, 0, 19.116, 73.118]
  MoveL 4198 to (-75.96, 0.35, -6.25) mm, rotated rx -180 ry 0 rz 90 deg; joints [73.082, -18.818, 89.685, 0, 19.133, 73.082]
  MoveC 4199 to (-74.74, -2.55, -6.25) mm, rotated rx 180 ry 0 rz 90 deg; joints [72.997, -18.787, 89.545, 0, 19.242, 72.997] to (-71.83, -3.76, -6.25) mm, rotated rx -180 ry 0 rz 90 deg; joints [72.986, -18.738, 89.325, 0, 19.412, 72.986]
  MoveC 4200 to (-70.91, -3.72, -6.25) mm, rotated rx 180 ry 0 rz 90 deg; joints [72.997, -18.724, 89.265, 0, 19.459, 72.997] to (-70, -3.56, -6.25) mm, rotated rx 180 ry 0 rz 90 deg; joints [73.012, -18.711, 89.207, 0, 19.504, 73.012]
  MoveL 4201 to (-20.9, 7.72, -6.25) mm, rotated rx 180 ry 0 rz 90 deg; joints [73.87, -17.967, 86.08, 0, 21.887, 73.87]
  MoveC 4202 to (-20.22, 7.92, -6.25) mm, rotated rx 180 ry 0 rz 90 deg; joints [73.882, -17.956, 86.037, 0, 21.919, 73.882] to (-19.57, 8.19, -6.25) mm, rotated rx -180 ry 0 rz 90 deg; joints [73.897, -17.946, 85.997, 0, 21.949, 73.897]
  MoveC 4203 to (-17.62, 10.14, -6.25) mm, rotated rx 180 ry 0 rz 90 deg; joints [73.98, -17.922, 85.9, 0, 22.022, 73.98] to (-17.36, 12.9, -6.25) mm, rotated rx -180 ry 0 rz 90 deg; joints [74.072, -17.931, 85.937, 0, 21.994, 74.072]
  MoveL 4204 to (-17.53, 13.55, -6.25) mm, rotated rx -180 ry 0 rz 90 deg; joints [74.092, -17.937, 85.962, 0, 21.975, 74.092]
  MoveL 4205 to (-17.59, 13.74, -6.25) mm, rotated rx 180 ry 0 rz 90 deg; joints [74.098, -17.939, 85.97, 0, 21.97, 74.098]
  MoveL 4206 to (-24.35, 32.63, -6.25) mm, rotated rx -180 ry 0 rz 90 deg; joints [74.658, -18.146, 86.808, 0, 21.338, 74.658]
  MoveC 4207 to (-25.08, 33.94, -6.25) mm, rotated rx 180 ry 0 rz 90 deg; joints [74.694, -18.164, 86.883, 0, 21.281, 74.694] to (-26.19, 34.95, -6.25) mm, rotated rx 180 ry 0 rz 90 deg; joints [74.718, -18.188, 86.979, 0, 21.209, 74.718]
  MoveL 4208 to (-68.47, 62.07, -6.25) mm, rotated rx -180 ry 0 rz 90 deg; joints [75.249, -18.966, 90.355, 0, 18.611, 75.249]
  MoveC 4209 to (-69.72, 62.75, -6.25) mm, rotated rx -180 ry 0 rz 90 deg; joints [75.261, -18.987, 90.451, 0, 18.536, 75.261] to (-71.07, 63.21, -6.25) mm, rotated rx -180 ry 0 rz 90 deg; joints [75.265, -19.008, 90.549, 0, 18.459, 75.265]
  MoveC 4210 to (-73.82, 62.74, -6.25) mm, rotated rx -180 ry 0 rz 90 deg; joints [75.224, -19.046, 90.725, 0, 18.321, 75.224] to (-75.68, 60.66, -6.25) mm, rotated rx 180 ry 0 rz 90 deg; joints [75.136, -19.065, 90.812, 0, 18.252, 75.136]
  MoveC 4211 to (-75.9, 59.73, -6.25) mm, rotated rx -180 ry 0 rz 90 deg; joints [75.102, -19.064, 90.81, 0, 18.254, 75.102] to (-75.97, 58.78, -6.25) mm, rotated rx 180 ry 0 rz 90 deg; joints [75.068, -19.062, 90.798, 0, 18.263, 75.068]
  MoveL 4212 to (-75.97, 29.57, -6.25) mm, rotated rx 180 ry 0 rz 90 deg; joints [74.07, -18.945, 90.261, 0, 18.685, 74.07]
  MoveL 4213 to (-68.42, 29.57, -6.25) mm, rotated rx 180 ry 0 rz 90 deg; joints [74.143, -18.834, 89.756, 0, 19.078, 74.143]
  MoveL 4214 to (-68.42, 29.57, -3.25) mm, rotated rx 180 ry 0 rz 90 deg; joints [74.143, -18.991, 89.857, 0, 19.134, 74.143]
  Establecer velocidad (1000.0 mm/s)
  MoveL 4215 to (-68.42, 29.57, 10) mm, rotated rx -180 ry 0 rz 90 deg; joints [74.143, -19.685, 90.299, 0, 19.386, 74.143]
  Establecer velocidad (66.7 mm/s)
  MoveL 4216 to (-67.52, 36.21, 10) mm, rotated rx -180 ry 0 rz 90 deg; joints [74.377, -19.699, 90.365, 0, 19.335, 74.377]
  MoveL 4217 to (-67.52, 36.21, -3.25) mm, rotated rx 180 ry 0 rz 90 deg; joints [74.377, -19.006, 89.923, 0, 19.083, 74.377]
  MoveL 4218 to (-69.03, 36.39, -3.66) mm, rotated rx -180 ry 0 rz 90 deg; joints [74.369, -19.008, 90.013, 0, 18.994, 74.369]
  MoveL 4219 to (-70.54, 36.21, -4.06) mm, rotated rx -180 ry 0 rz 90 deg; joints [74.348, -19.008, 90.097, 0, 18.911, 74.348]
  MoveL 4220 to (-71.97, 35.7, -4.47) mm, rotated rx -180 ry 0 rz 90 deg; joints [74.317, -19.006, 90.17, 0, 18.836, 74.317]
  MoveL 4221 to (-73.25, 34.88, -4.87) mm, rotated rx 180 ry 0 rz 90 deg; joints [74.277, -19, 90.226, 0, 18.774, 74.277]
  MoveL 4222 to (-74.32, 33.8, -5.28) mm, rotated rx 180 ry 0 rz 90 deg; joints [74.23, -18.99, 90.264, 0, 18.726, 74.23]
  MoveL 4223 to (-75.13, 32.51, -5.69) mm, rotated rx -180 ry 0 rz 90 deg; joints [74.179, -18.975, 90.279, 0, 18.696, 74.179]
  MoveL 4224 to (-75.62, 31.08, -6.09) mm, rotated rx 180 ry 0 rz 90 deg; joints [74.125, -18.955, 90.272, 0, 18.683, 74.125]
  MoveL 4225 to (-75.76, 29.57, -6.5) mm, rotated rx 180 ry 0 rz 90 deg; joints [74.072, -18.929, 90.239, 0, 18.691, 74.072]
  MoveL 4226 to (-75.76, 1.42, -6.5) mm, rotated rx 180 ry 0 rz 90 deg; joints [73.12, -18.807, 89.686, 0, 19.122, 73.12]
  MoveL 4227 to (-75.75, 0.47, -6.5) mm, rotated rx 180 ry 0 rz 90 deg; joints [73.089, -18.803, 89.666, 0, 19.137, 73.089]
  MoveC 4228 to (-74.53, -2.44, -6.5) mm, rotated rx 180 ry 0 rz 90 deg; joints [73.003, -18.771, 89.524, 0, 19.247, 73.003] to (-71.56, -3.55, -6.5) mm, rotated rx -180 ry 0 rz 90 deg; joints [72.996, -18.722, 89.303, 0, 19.418, 72.996]
  MoveC 4229 to (-70.8, -3.48, -6.5) mm, rotated rx -180 ry 0 rz 90 deg; joints [73.007, -18.71, 89.254, 0, 19.457, 73.007] to (-70.05, -3.35, -6.5) mm, rotated rx 180 ry 0 rz 90 deg; joints [73.019, -18.699, 89.206, 0, 19.494, 73.019]
  MoveL 4230 to (-68.7, -3.06, -6.5) mm, rotated rx 180 ry 0 rz 90 deg; joints [73.042, -18.68, 89.122, 0, 19.559, 73.042]
  MoveL 4231 to (-21.32, 7.85, -6.5) mm, rotated rx 180 ry 0 rz 90 deg; joints [73.869, -17.962, 86.104, 0, 21.858, 73.869]
  MoveC 4232 to (-20.68, 8.01, -6.5) mm, rotated rx 180 ry 0 rz 90 deg; joints [73.881, -17.951, 86.062, 0, 21.89, 73.881] to (-20.04, 8.21, -6.5) mm, rotated rx -180 ry 0 rz 90 deg; joints [73.894, -17.941, 86.022, 0, 21.92, 73.894]
  MoveC 4233 to (-18, 9.91, -6.5) mm, rotated rx 180 ry 0 rz 90 deg; joints [73.968, -17.914, 85.914, 0, 22.001, 73.968] to (-17.51, 12.51, -6.5) mm, rotated rx 180 ry 0 rz 90 deg; joints [74.058, -17.919, 85.931, 0, 21.988, 74.058]
  MoveC 4234 to (-17.67, 13.28, -6.5) mm, rotated rx -180 ry 0 rz 90 deg; joints [74.082, -17.925, 85.958, 0, 21.968, 74.082] to (-17.9, 14.03, -6.5) mm, rotated rx 180 ry 0 rz 90 deg; joints [74.104, -17.933, 85.988, 0, 21.945, 74.104]
  MoveL 4235 to (-24.51, 32.5, -6.5) mm, rotated rx 180 ry 0 rz 90 deg; joints [74.652, -18.135, 86.808, 0, 21.327, 74.652]
  MoveC 4236 to (-25.25, 33.83, -6.5) mm, rotated rx 180 ry 0 rz 90 deg; joints [74.689, -18.154, 86.885, 0, 21.269, 74.689] to (-26.39, 34.85, -6.5) mm, rotated rx 180 ry 0 rz 90 deg; joints [74.713, -18.178, 86.983, 0, 21.195, 74.713]
  MoveL 4237 to (-68.56, 61.91, -6.5) mm, rotated rx -180 ry 0 rz 90 deg; joints [75.243, -18.954, 90.35, 0, 18.603, 75.243]
  MoveC 4238 to (-69.55, 62.45, -6.5) mm, rotated rx 180 ry 0 rz 90 deg; joints [75.252, -18.97, 90.426, 0, 18.544, 75.252] to (-70.6, 62.85, -6.5) mm, rotated rx -180 ry 0 rz 90 deg; joints [75.257, -18.987, 90.503, 0, 18.484, 75.257]
  MoveC 4239 to (-73.64, 62.53, -6.5) mm, rotated rx -180 ry 0 rz 90 deg; joints [75.218, -19.03, 90.701, 0, 18.329, 75.218] to (-75.59, 60.18, -6.5) mm, rotated rx 180 ry 0 rz 90 deg; joints [75.12, -19.049, 90.789, 0, 18.259, 75.12]
  MoveC 4240 to (-75.72, 59.62, -6.5) mm, rotated rx -180 ry 0 rz 90 deg; joints [75.099, -19.048, 90.788, 0, 18.26, 75.099] to (-75.76, 59.05, -6.5) mm, rotated rx -180 ry 0 rz 90 deg; joints [75.079, -19.047, 90.781, 0, 18.266, 75.079]
  MoveL 4241 to (-75.76, 29.57, -6.5) mm, rotated rx 180 ry 0 rz 90 deg; joints [74.072, -18.929, 90.239, 0, 18.691, 74.072]
  MoveL 4242 to (-68.21, 29.57, -6.5) mm, rotated rx 180 ry 0 rz 90 deg; joints [74.145, -18.818, 89.734, 0, 19.084, 74.145]
  MoveL 4243 to (-68.21, 29.57, -3.5) mm, rotated rx 180 ry 0 rz 90 deg; joints [74.145, -18.975, 89.835, 0, 19.14, 74.145]
  Establecer velocidad (1000.0 mm/s)
  MoveL 4244 to (-68.21, 29.57, 10) mm, rotated rx -180 ry 0 rz 90 deg; joints [74.145, -19.681, 90.285, 0, 19.396, 74.145]
  Establecer velocidad (66.7 mm/s)
  MoveL 4245 to (-39.61, -29.7, 10) mm, rotated rx 180 ry 0 rz 90 deg; joints [72.46, -18.931, 87.134, 0, 21.797, 72.46]
  MoveL 4246 to (-39.61, -29.7, -3.25) mm, rotated rx -180 ry 0 rz 90 deg; joints [72.46, -18.248, 86.693, 0, 21.555, 72.46]
  MoveL 4247 to (-39.74, -28.19, -3.66) mm, rotated rx 180 ry 0 rz 90 deg; joints [72.508, -18.237, 86.721, 0, 21.516, 72.508]
  MoveL 4248 to (-40.24, -26.75, -4.06) mm, rotated rx -180 ry 0 rz 90 deg; joints [72.55, -18.232, 86.772, 0, 21.46, 72.55]
  MoveL 4249 to (-41.03, -25.46, -4.47) mm, rotated rx 180 ry 0 rz 90 deg; joints [72.584, -18.232, 86.841, 0, 21.39, 72.584]
  MoveL 4250 to (-42.1, -24.37, -4.87) mm, rotated rx 180 ry 0 rz 90 deg; joints [72.609, -18.234, 86.924, 0, 21.31, 72.609]
  MoveL 4251 to (-43.38, -23.55, -5.28) mm, rotated rx 180 ry 0 rz 90 deg; joints [72.622, -18.239, 87.015, 0, 21.223, 72.622]
  MoveL 4252 to (-44.81, -23.03, -5.69) mm, rotated rx 180 ry 0 rz 90 deg; joints [72.625, -18.244, 87.111, 0, 21.133, 72.625]
  MoveL 4253 to (-46.31, -22.84, -6.09) mm, rotated rx 180 ry 0 rz 90 deg; joints [72.615, -18.249, 87.204, 0, 21.045, 72.615]
  MoveL 4254 to (-47.82, -23.02, -6.5) mm, rotated rx 180 ry 0 rz 90 deg; joints [72.594, -18.252, 87.289, 0, 20.962, 72.594]
  MoveL 4255 to (-72.42, -28.25, -6.5) mm, rotated rx 180 ry 0 rz 90 deg; joints [72.163, -18.616, 88.841, 0, 19.775, 72.163]
  MoveC 4256 to (-74.82, -29.73, -6.5) mm, rotated rx -180 ry 0 rz 90 deg; joints [72.088, -18.646, 88.97, 0, 19.676, 72.088] to (-75.76, -32.38, -6.5) mm, rotated rx -180 ry 0 rz 90 deg; joints [71.99, -18.647, 88.976, 0, 19.672, 71.99]
  MoveL 4257 to (-75.76, -71.02, -6.5) mm, rotated rx -180 ry 0 rz 90 deg; joints [70.715, -18.445, 88.103, 0, 20.342, 70.715]
  MoveC 4258 to (-74.99, -73.38, -6.5) mm, rotated rx -180 ry 0 rz 90 deg; joints [70.646, -18.42, 87.996, 0, 20.424, 70.646] to (-72.98, -74.84, -6.5) mm, rotated rx 180 ry 0 rz 90 deg; joints [70.622, -18.38, 87.827, 0, 20.553, 70.622]
  MoveC 4259 to (-72.08, -75.06, -6.5) mm, rotated rx 180 ry 0 rz 90 deg; joints [70.625, -18.365, 87.761, 0, 20.603, 70.625] to (-71.16, -75.12, -6.5) mm, rotated rx 180 ry 0 rz 90 deg; joints [70.633, -18.35, 87.698, 0, 20.652, 70.633]
  MoveL 4260 to (-35.28, -74.85, -6.5) mm, rotated rx -180 ry 0 rz 90 deg; joints [71.045, -17.749, 85.257, 0, 22.492, 71.045]
  MoveC 4261 to (-33.16, -74.24, -6.5) mm, rotated rx 180 ry 0 rz 90 deg; joints [71.088, -17.715, 85.125, 0, 22.591, 71.088] to (-31.64, -72.64, -6.5) mm, rotated rx 180 ry 0 rz 90 deg; joints [71.156, -17.698, 85.057, 0, 22.641, 71.156]
  MoveC 4262 to (-31.32, -71.95, -6.5) mm, rotated rx -180 ry 0 rz 90 deg; joints [71.181, -17.697, 85.052, 0, 22.645, 71.181] to (-31.09, -71.23, -6.5) mm, rotated rx 180 ry 0 rz 90 deg; joints [71.207, -17.697, 85.052, 0, 22.644, 71.207]
  MoveL 4263 to (-18.66, -23.57, -6.5) mm, rotated rx -180 ry 0 rz 90 deg; joints [72.872, -17.75, 85.263, 0, 22.487, 72.872]
  MoveC 4264 to (-18.45, -22.46, -6.5) mm, rotated rx 180 ry 0 rz 90 deg; joints [72.91, -17.753, 85.272, 0, 22.48, 72.91] to (-18.4, -21.32, -6.5) mm, rotated rx -180 ry 0 rz 90 deg; joints [72.947, -17.758, 85.293, 0, 22.465, 72.947]
  MoveC 4265 to (-19.55, -19, -6.5) mm, rotated rx -180 ry 0 rz 90 deg; joints [73.011, -17.791, 85.423, 0, 22.368, 73.011] to (-21.8, -17.72, -6.5) mm, rotated rx -180 ry 0 rz 90 deg; joints [73.03, -17.838, 85.607, 0, 22.23, 73.03]
  MoveC 4266 to (-22.51, -17.7, -6.5) mm, rotated rx 180 ry 0 rz 90 deg; joints [73.024, -17.85, 85.657, 0, 22.193, 73.024] to (-23.22, -17.79, -6.5) mm, rotated rx 180 ry 0 rz 90 deg; joints [73.014, -17.862, 85.705, 0, 22.157, 73.014]
  MoveL 4267 to (-47.82, -23.02, -6.5) mm, rotated rx 180 ry 0 rz 90 deg; joints [72.594, -18.252, 87.289, 0, 20.962, 72.594]
  MoveL 4268 to (-46.25, -30.41, -6.5) mm, rotated rx -180 ry 0 rz 90 deg; joints [72.368, -18.187, 87.023, 0, 21.165, 72.368]
  MoveL 4269 to (-46.25, -30.41, -3.5) mm, rotated rx 180 ry 0 rz 90 deg; joints [72.368, -18.343, 87.124, 0, 21.218, 72.368]
  Establecer velocidad (1000.0 mm/s)
  MoveL 4270 to (-46.25, -30.41, 10) mm, rotated rx 180 ry 0 rz 90 deg; joints [72.368, -19.04, 87.574, 0, 21.466, 72.368]
  Establecer velocidad (66.7 mm/s)
  MoveL 4271 to (17.17, -66.59, 10) mm, rotated rx 180 ry 0 rz 90 deg; joints [71.864, -17.652, 82.299, 0, 25.353, 71.864]
  MoveL 4272 to (17.17, -66.59, -3.25) mm, rotated rx 180 ry 0 rz 90 deg; joints [71.864, -16.982, 81.856, 0, 25.126, 71.864]
  MoveL 4273 to (17, -68.1, -3.66) mm, rotated rx 180 ry 0 rz 90 deg; joints [71.815, -16.955, 81.818, 0, 25.137, 71.815]
  MoveL 4274 to (17.21, -69.61, -4.06) mm, rotated rx -180 ry 0 rz 90 deg; joints [71.77, -16.92, 81.754, 0, 25.167, 71.77]
  MoveL 4275 to (17.74, -71.03, -4.47) mm, rotated rx -180 ry 0 rz 90 deg; joints [71.731, -16.88, 81.668, 0, 25.212, 71.731]
  MoveL 4276 to (18.57, -72.3, -4.87) mm, rotated rx -180 ry 0 rz 90 deg; joints [71.7, -16.834, 81.563, 0, 25.271, 71.7]
  MoveL 4277 to (19.66, -73.36, -5.28) mm, rotated rx -180 ry 0 rz 90 deg; joints [71.679, -16.784, 81.445, 0, 25.339, 71.679]
  MoveL 4278 to (20.97, -74.14, -5.69) mm, rotated rx -180 ry 0 rz 90 deg; joints [71.668, -16.732, 81.318, 0, 25.414, 71.668]
  MoveL 4279 to (22.41, -74.62, -6.09) mm, rotated rx 180 ry 0 rz 90 deg; joints [71.667, -16.679, 81.188, 0, 25.491, 71.667]
  MoveL 4280 to (23.92, -74.74, -6.5) mm, rotated rx 180 ry 0 rz 90 deg; joints [71.679, -16.627, 81.061, 0, 25.566, 71.679]
  MoveC 4281 to (36.83, -74.54, -6.5) mm, rotated rx 180 ry 0 rz 90 deg; joints [71.818, -16.362, 80.121, 0, 26.24, 71.818] to (49.75, -74.31, -6.5) mm, rotated rx -180 ry 0 rz 90 deg; joints [71.955, -16.088, 79.171, 0, 26.917, 71.955]
  MoveC 4282 to (52.48, -71.19, -6.5) mm, rotated rx -180 ry 0 rz 90 deg; joints [72.078, -16.051, 79.043, 0, 27.008, 72.078] to (52.59, -67.05, -6.5) mm, rotated rx -180 ry 0 rz 90 deg; joints [72.207, -16.077, 79.134, 0, 26.944, 72.207]
  MoveL 4283 to (49.97, -63.97, -6.5) mm, rotated rx -180 ry 0 rz 90 deg; joints [72.276, -16.155, 79.402, 0, 26.753, 72.276]
  MoveL 4284 to (26.38, -36.48, -6.5) mm, rotated rx 180 ry 0 rz 90 deg; joints [72.902, -16.824, 81.771, 0, 25.054, 72.902]
  MoveC 4285 to (25.77, -35.86, -6.5) mm, rotated rx 180 ry 0 rz 90 deg; joints [72.916, -16.84, 81.828, 0, 25.012, 72.916] to (25.11, -35.3, -6.5) mm, rotated rx 180 ry 0 rz 90 deg; joints [72.928, -16.857, 81.889, 0, 24.968, 72.928]
  MoveL 4286 to (12.39, -25.11, -6.5) mm, rotated rx -180 ry 0 rz 90 deg; joints [73.127, -17.167, 83.031, 0, 24.136, 73.127]
  MoveL 4287 to (11.85, -24.67, -6.5) mm, rotated rx 180 ry 0 rz 90 deg; joints [73.136, -17.18, 83.08, 0, 24.1, 73.136]
  MoveC 4288 to (8.81, -24.18, -6.5) mm, rotated rx 180 ry 0 rz 90 deg; joints [73.122, -17.241, 83.308, 0, 23.933, 73.122] to (6.16, -25.74, -6.5) mm, rotated rx -180 ry 0 rz 90 deg; joints [73.047, -17.282, 83.463, 0, 23.819, 73.047]
  MoveC 4289 to (5.88, -26.16, -6.5) mm, rotated rx -180 ry 0 rz 90 deg; joints [73.031, -17.285, 83.474, 0, 23.811, 73.031] to (5.7, -26.63, -6.5) mm, rotated rx -180 ry 0 rz 90 deg; joints [73.014, -17.286, 83.477, 0, 23.809, 73.014]
  MoveL 4290 to (-5.84, -69.97, -6.5) mm, rotated rx 180 ry 0 rz 90 deg; joints [71.518, -17.242, 83.312, 0, 23.93, 71.518]
  MoveC 4291 to (-5.13, -73.47, -6.5) mm, rotated rx 180 ry 0 rz 90 deg; joints [71.415, -17.207, 83.178, 0, 24.028, 71.415] to (-1.91, -75.03, -6.5) mm, rotated rx 180 ry 0 rz 90 deg; joints [71.4, -17.135, 82.912, 0, 24.223, 71.4]
  MoveC 4292 to (11, -74.9, -6.5) mm, rotated rx 180 ry 0 rz 90 deg; joints [71.54, -16.885, 81.991, 0, 24.894, 71.54] to (23.92, -74.74, -6.5) mm, rotated rx 180 ry 0 rz 90 deg; joints [71.679, -16.627, 81.061, 0, 25.566, 71.679]
  MoveL 4293 to (23.81, -67.19, -6.5) mm, rotated rx 180 ry 0 rz 90 deg; joints [71.914, -16.68, 81.249, 0, 25.43, 71.914]
  MoveL 4294 to (23.81, -67.19, -3.5) mm, rotated rx 180 ry 0 rz 90 deg; joints [71.914, -16.831, 81.351, 0, 25.48, 71.914]
  Establecer velocidad (1000.0 mm/s)
  MoveL 4295 to (23.81, -67.19, 10) mm, rotated rx 180 ry 0 rz 90 deg; joints [71.914, -17.513, 81.804, 0, 25.709, 71.914]
  Establecer velocidad (66.7 mm/s)
  MoveL 4296 to (64.78, -31.42, 10) mm, rotated rx -180 ry 0 rz 90 deg; joints [73.424, -16.879, 79.603, 0, 27.276, 73.424]
  MoveL 4297 to (64.78, -31.42, -3.25) mm, rotated rx 180 ry 0 rz 90 deg; joints [73.424, -16.215, 79.158, 0, 27.058, 73.424]
  MoveL 4298 to (66.28, -31.61, -3.66) mm, rotated rx -180 ry 0 rz 90 deg; joints [73.432, -16.161, 79.027, 0, 27.134, 73.432]
  MoveL 4299 to (67.79, -31.42, -4.06) mm, rotated rx 180 ry 0 rz 90 deg; joints [73.451, -16.108, 78.903, 0, 27.205, 73.451]
  MoveL 4300 to (69.22, -30.91, -4.47) mm, rotated rx -180 ry 0 rz 90 deg; joints [73.48, -16.06, 78.793, 0, 27.267, 73.48]
  MoveL 4301 to (70.5, -30.09, -4.87) mm, rotated rx -180 ry 0 rz 90 deg; joints [73.517, -16.016, 78.701, 0, 27.316, 73.517]
  MoveL 4302 to (71.57, -29.01, -5.28) mm, rotated rx 180 ry 0 rz 90 deg; joints [73.56, -15.979, 78.63, 0, 27.349, 73.56]
  MoveL 4303 to (72.37, -27.73, -5.69) mm, rotated rx -180 ry 0 rz 90 deg; joints [73.607, -15.949, 78.584, 0, 27.366, 73.607]
  MoveL 4304 to (72.88, -26.29, -6.09) mm, rotated rx -180 ry 0 rz 90 deg; joints [73.656, -15.927, 78.564, 0, 27.363, 73.656]
  MoveL 4305 to (73.01, -24.78, -6.5) mm, rotated rx 180 ry 0 rz 90 deg; joints [73.704, -15.914, 78.573, 0, 27.341, 73.704]
  MoveL 4306 to (73.01, -11.72, -6.5) mm, rotated rx -180 ry 0 rz 90 deg; joints [74.109, -15.997, 78.858, 0, 27.139, 74.109]
  MoveC 4307 to (71.28, -9.21, -6.5) mm, rotated rx 180 ry 0 rz 90 deg; joints [74.171, -16.051, 79.043, 0, 27.008, 74.171] to (68.67, -7.6, -6.5) mm, rotated rx 180 ry 0 rz 90 deg; joints [74.198, -16.118, 79.274, 0, 26.844, 74.198]
  MoveC 4308 to (67.15, -7.32, -6.5) mm, rotated rx 180 ry 0 rz 90 deg; joints [74.194, -16.153, 79.394, 0, 26.759, 74.194] to (65.63, -7.53, -6.5) mm, rotated rx 180 ry 0 rz 90 deg; joints [74.174, -16.185, 79.504, 0, 26.681, 74.174]
  MoveL 4309 to (65.39, -7.86, -6.5) mm, rotated rx -180 ry 0 rz 90 deg; joints [74.162, -16.188, 79.515, 0, 26.673, 74.162]
  MoveL 4310 to (56.23, -20.37, -6.5) mm, rotated rx -180 ry 0 rz 90 deg; joints [73.689, -16.307, 79.93, 0, 26.377, 73.689]
  MoveL 4311 to (53.87, -23.57, -6.5) mm, rotated rx 180 ry 0 rz 90 deg; joints [73.567, -16.337, 80.036, 0, 26.302, 73.567]
  MoveC 4312 to (53.27, -24.75, -6.5) mm, rotated rx -180 ry 0 rz 90 deg; joints [73.525, -16.343, 80.055, 0, 26.288, 73.525] to (53.07, -26.06, -6.5) mm, rotated rx -180 ry 0 rz 90 deg; joints [73.482, -16.338, 80.04, 0, 26.298, 73.482]
  MoveC 4313 to (53.39, -27.42, -6.5) mm, rotated rx 180 ry 0 rz 90 deg; joints [73.443, -16.323, 79.987, 0, 26.336, 73.443] to (54.13, -28.6, -6.5) mm, rotated rx -180 ry 0 rz 90 deg; joints [73.413, -16.3, 79.905, 0, 26.395, 73.413]
  MoveL 4314 to (55.26, -29.85, -6.5) mm, rotated rx 180 ry 0 rz 90 deg; joints [73.384, -16.268, 79.794, 0, 26.474, 73.384]
  MoveL 4315 to (66.03, -41.97, -6.5) mm, rotated rx 180 ry 0 rz 90 deg; joints [73.109, -15.955, 78.713, 0, 27.241, 73.109]
  MoveC 4316 to (68.27, -42.03, -6.5) mm, rotated rx -180 ry 0 rz 90 deg; joints [73.128, -15.905, 78.543, 0, 27.362, 73.128] to (70.34, -41.17, -6.5) mm, rotated rx 180 ry 0 rz 90 deg; joints [73.174, -15.865, 78.406, 0, 27.458, 73.174]
  MoveC 4317 to (71.92, -39.7, -6.5) mm, rotated rx -180 ry 0 rz 90 deg; joints [73.234, -15.839, 78.32, 0, 27.519, 73.234] to (73.01, -37.84, -6.5) mm, rotated rx 180 ry 0 rz 90 deg; joints [73.301, -15.828, 78.28, 0, 27.547, 73.301]
  MoveL 4318 to (73.01, -24.78, -6.5) mm, rotated rx 180 ry 0 rz 90 deg; joints [73.704, -15.914, 78.573, 0, 27.341, 73.704]
  MoveL 4319 to (65.46, -24.78, -6.5) mm, rotated rx 180 ry 0 rz 90 deg; joints [73.636, -16.08, 79.142, 0, 26.937, 73.636]
  MoveL 4320 to (65.46, -24.78, -3.5) mm, rotated rx -180 ry 0 rz 90 deg; joints [73.636, -16.231, 79.245, 0, 26.986, 73.636]
  Establecer velocidad (1000.0 mm/s)
  MoveL 4321 to (65.46, -24.78, 10) mm, rotated rx 180 ry 0 rz 90 deg; joints [73.636, -16.907, 79.699, 0, 27.208, 73.636]
  Establecer velocidad (66.7 mm/s)
  MoveL 4322 to (36.75, 22.16, 10) mm, rotated rx 180 ry 0 rz 90 deg; joints [74.858, -17.792, 82.802, 0, 24.989, 74.858]
  MoveL 4323 to (36.75, 22.16, -3.25) mm, rotated rx 180 ry 0 rz 90 deg; joints [74.858, -17.12, 82.359, 0, 24.761, 74.858]
  MoveL 4324 to (36.91, 23.67, -3.66) mm, rotated rx -180 ry 0 rz 90 deg; joints [74.908, -17.105, 82.364, 0, 24.741, 74.908]
  MoveL 4325 to (36.69, 25.17, -4.06) mm, rotated rx 180 ry 0 rz 90 deg; joints [74.954, -17.097, 82.396, 0, 24.701, 74.954]
  MoveL 4326 to (36.14, 26.59, -4.47) mm, rotated rx -180 ry 0 rz 90 deg; joints [74.995, -17.095, 82.45, 0, 24.645, 74.995]
  MoveL 4327 to (35.3, 27.85, -4.87) mm, rotated rx -180 ry 0 rz 90 deg; joints [75.028, -17.097, 82.522, 0, 24.575, 75.028]
  MoveL 4328 to (34.19, 28.9, -5.28) mm, rotated rx 180 ry 0 rz 90 deg; joints [75.052, -17.104, 82.609, 0, 24.495, 75.052]
  MoveL 4329 to (32.89, 29.67, -5.69) mm, rotated rx -180 ry 0 rz 90 deg; joints [75.066, -17.113, 82.706, 0, 24.408, 75.066]
  MoveL 4330 to (31.44, 30.13, -6.09) mm, rotated rx 180 ry 0 rz 90 deg; joints [75.068, -17.124, 82.806, 0, 24.317, 75.068]
  MoveL 4331 to (29.93, 30.24, -6.5) mm, rotated rx -180 ry 0 rz 90 deg; joints [75.059, -17.133, 82.904, 0, 24.229, 75.059]
  MoveL 4332 to (9, 29.75, -6.5) mm, rotated rx -180 ry 0 rz 90 deg; joints [74.861, -17.528, 84.399, 0, 23.129, 74.861]
  MoveC 4333 to (6.03, 28.02, -6.5) mm, rotated rx 180 ry 0 rz 90 deg; joints [74.779, -17.575, 84.577, 0, 22.997, 74.779] to (5.37, 24.64, -6.5) mm, rotated rx 180 ry 0 rz 90 deg; joints [74.663, -17.57, 84.559, 0, 23.011, 74.663]
  MoveL 4334 to (5.54, 24.17, -6.5) mm, rotated rx -180 ry 0 rz 90 deg; joints [74.649, -17.564, 84.537, 0, 23.027, 74.649]
  MoveL 4335 to (10.36, 10.9, -6.5) mm, rotated rx 180 ry 0 rz 90 deg; joints [74.263, -17.406, 83.931, 0, 23.475, 74.263]
  MoveL 4336 to (10.99, 9.15, -6.5) mm, rotated rx 180 ry 0 rz 90 deg; joints [74.212, -17.385, 83.85, 0, 23.535, 74.212]
  MoveC 4337 to (11.54, 8.12, -6.5) mm, rotated rx 180 ry 0 rz 90 deg; joints [74.184, -17.369, 83.79, 0, 23.579, 74.184] to (12.35, 7.29, -6.5) mm, rotated rx 180 ry 0 rz 90 deg; joints [74.165, -17.349, 83.715, 0, 23.634, 74.165]
  MoveL 4338 to (28.32, -5.04, -6.5) mm, rotated rx -180 ry 0 rz 90 deg; joints [73.916, -16.972, 82.31, 0, 24.662, 73.916]
  MoveC 4339 to (29.62, -5.68, -6.5) mm, rotated rx -180 ry 0 rz 90 deg; joints [73.908, -16.943, 82.202, 0, 24.741, 73.908] to (31.07, -5.77, -6.5) mm, rotated rx 180 ry 0 rz 90 deg; joints [73.918, -16.913, 82.095, 0, 24.819, 73.918]
  MoveL 4340 to (31.41, -5.73, -6.5) mm, rotated rx -180 ry 0 rz 90 deg; joints [73.923, -16.907, 82.071, 0, 24.836, 73.923]
  MoveC 4341 to (33.02, -5.16, -6.5) mm, rotated rx 180 ry 0 rz 90 deg; joints [73.955, -16.878, 81.966, 0, 24.912, 73.955] to (34.27, -4, -6.5) mm, rotated rx -180 ry 0 rz 90 deg; joints [74.004, -16.859, 81.899, 0, 24.961, 74.004]
  MoveL 4342 to (52.59, 21.71, -6.5) mm, rotated rx 180 ry 0 rz 90 deg; joints [74.98, -16.631, 81.076, 0, 25.555, 74.98]
  MoveL 4343 to (53.99, 23.69, -6.5) mm, rotated rx 180 ry 0 rz 90 deg; joints [75.054, -16.613, 81.012, 0, 25.601, 75.054]
  MoveC 4344 to (53.71, 27.76, -6.5) mm, rotated rx 180 ry 0 rz 90 deg; joints [75.181, -16.642, 81.113, 0, 25.529, 75.181] to (50.85, 30.68, -6.5) mm, rotated rx -180 ry 0 rz 90 deg; joints [75.25, -16.716, 81.381, 0, 25.335, 75.25]
  MoveL 4345 to (45.96, 30.61, -6.5) mm, rotated rx -180 ry 0 rz 90 deg; joints [75.207, -16.816, 81.74, 0, 25.076, 75.207]
  MoveL 4346 to (29.93, 30.24, -6.5) mm, rotated rx -180 ry 0 rz 90 deg; joints [75.059, -17.133, 82.904, 0, 24.229, 75.059]
  MoveL 4347 to (30.1, 22.69, -6.5) mm, rotated rx 180 ry 0 rz 90 deg; joints [74.818, -17.09, 82.744, 0, 24.346, 74.818]
  MoveL 4348 to (30.1, 22.69, -3.5) mm, rotated rx 180 ry 0 rz 90 deg; joints [74.818, -17.242, 82.846, 0, 24.397, 74.818]
  Establecer velocidad (1000.0 mm/s)
  MoveL 4349 to (30.1, 22.69, 10) mm, rotated rx -180 ry 0 rz 90 deg; joints [74.818, -17.928, 83.297, 0, 24.631, 74.818]
  Establecer velocidad (66.7 mm/s)
  MoveL 4350 to (26.9, 66.26, 10) mm, rotated rx 180 ry 0 rz 90 deg; joints [76.198, -18.21, 84.343, 0, 23.867, 76.198]
  MoveL 4351 to (26.9, 66.26, -3.25) mm, rotated rx -180 ry 0 rz 90 deg; joints [76.198, -17.535, 83.901, 0, 23.634, 76.198]
  MoveL 4352 to (27.1, 67.76, -3.66) mm, rotated rx -180 ry 0 rz 90 deg; joints [76.248, -17.518, 83.899, 0, 23.618, 76.248]
  MoveL 4353 to (26.94, 69.27, -4.06) mm, rotated rx 180 ry 0 rz 90 deg; joints [76.296, -17.507, 83.924, 0, 23.583, 76.296]
  MoveL 4354 to (26.45, 70.71, -4.47) mm, rotated rx 180 ry 0 rz 90 deg; joints [76.339, -17.502, 83.971, 0, 23.532, 76.339]
  MoveL 4355 to (25.65, 72, -4.87) mm, rotated rx 180 ry 0 rz 90 deg; joints [76.375, -17.502, 84.037, 0, 23.466, 76.375]
  MoveL 4356 to (24.59, 73.09, -5.28) mm, rotated rx 180 ry 0 rz 90 deg; joints [76.402, -17.507, 84.119, 0, 23.388, 76.402]
  MoveL 4357 to (23.31, 73.91, -5.69) mm, rotated rx 180 ry 0 rz 90 deg; joints [76.419, -17.514, 84.211, 0, 23.303, 76.419]
  MoveL 4358 to (21.88, 74.43, -6.09) mm, rotated rx 180 ry 0 rz 90 deg; joints [76.425, -17.522, 84.309, 0, 23.213, 76.425]
  MoveL 4359 to (20.38, 74.59, -6.5) mm, rotated rx -180 ry 0 rz 90 deg; joints [76.418, -17.53, 84.407, 0, 23.124, 76.418]
  MoveL 4360 to (12.79, 74.7, -6.5) mm, rotated rx 180 ry 0 rz 90 deg; joints [76.361, -17.671, 84.951, 0, 22.72, 76.361]
  MoveL 4361 to (-28.43, 75.15, -6.5) mm, rotated rx -180 ry 0 rz 90 deg; joints [76.04, -18.386, 87.851, 0, 20.535, 76.04]
  MoveC 4362 to (-31.04, 71.8, -6.5) mm, rotated rx 180 ry 0 rz 90 deg; joints [75.905, -18.415, 87.974, 0, 20.441, 75.905] to (-30.59, 67.57, -6.5) mm, rotated rx 180 ry 0 rz 90 deg; joints [75.767, -18.39, 87.869, 0, 20.521, 75.767]
  MoveL 4363 to (-10.56, 54.85, -6.5) mm, rotated rx -180 ry 0 rz 90 deg; joints [75.514, -17.998, 86.251, 0, 21.748, 75.514]
  MoveC 4364 to (-8.93, 54.15, -6.5) mm, rotated rx 180 ry 0 rz 90 deg; joints [75.505, -17.967, 86.124, 0, 21.843, 75.505] to (-7.16, 54, -6.5) mm, rotated rx -180 ry 0 rz 90 deg; joints [75.515, -17.935, 85.997, 0, 21.939, 75.515]
  MoveL 4365 to (35.54, 57.18, -6.5) mm, rotated rx -180 ry 0 rz 90 deg; joints [75.973, -17.159, 83.002, 0, 24.157, 75.973]
  MoveL 4366 to (39.33, 57.49, -6.5) mm, rotated rx -180 ry 0 rz 90 deg; joints [76.013, -17.086, 82.731, 0, 24.355, 76.013]
  MoveC 4367 to (54.31, 58.87, -6.5) mm, rotated rx 180 ry 0 rz 90 deg; joints [76.177, -16.793, 81.656, 0, 25.137, 76.177] to (69.26, 60.61, -6.5) mm, rotated rx -180 ry 0 rz 90 deg; joints [76.349, -16.491, 80.575, 0, 25.915, 76.349]
  MoveC 4368 to (71.32, 61.71, -6.5) mm, rotated rx 180 ry 0 rz 90 deg; joints [76.4, -16.453, 80.441, 0, 26.011, 76.4] to (72.14, 63.89, -6.5) mm, rotated rx -180 ry 0 rz 90 deg; joints [76.475, -16.446, 80.419, 0, 26.027, 76.475]
  MoveL 4369 to (72.14, 69.75, -6.5) mm, rotated rx -180 ry 0 rz 90 deg; joints [76.661, -16.476, 80.524, 0, 25.952, 76.661]
  MoveC 4370 to (71.28, 71.92, -6.5) mm, rotated rx -180 ry 0 rz 90 deg; joints [76.724, -16.505, 80.627, 0, 25.878, 76.724] to (69.15, 72.91, -6.5) mm, rotated rx 180 ry 0 rz 90 deg; joints [76.739, -16.555, 80.804, 0, 25.751, 76.739]
  MoveC 4371 to (45.25, 74.01, -6.5) mm, rotated rx -180 ry 0 rz 90 deg; joints [76.593, -17.049, 82.593, 0, 24.456, 76.593] to (21.32, 74.58, -6.5) mm, rotated rx 180 ry 0 rz 90 deg; joints [76.425, -17.513, 84.338, 0, 23.174, 76.425]
  MoveL 4372 to (20.38, 74.59, -6.5) mm, rotated rx -180 ry 0 rz 90 deg; joints [76.418, -17.53, 84.407, 0, 23.124, 76.418]
  MoveL 4373 to (20.27, 67.04, -6.5) mm, rotated rx 180 ry 0 rz 90 deg; joints [76.17, -17.498, 84.282, 0, 23.216, 76.17]
  MoveL 4374 to (20.27, 67.04, -3.5) mm, rotated rx 180 ry 0 rz 90 deg; joints [76.17, -17.651, 84.384, 0, 23.268, 76.17]
  Establecer velocidad (1000.0 mm/s)
  MoveL 4375 to (20.27, 67.04, 10) mm, rotated rx 180 ry 0 rz 90 deg; joints [76.17, -18.341, 84.834, 0, 23.507, 76.17]
  Establecer velocidad (66.7 mm/s)
  MoveL 4376 to (26.87, 65.99, 10) mm, rotated rx -180 ry 0 rz 90 deg; joints [76.189, -18.21, 84.341, 0, 23.869, 76.189]
  MoveL 4377 to (26.87, 65.99, -3.5) mm, rotated rx 180 ry 0 rz 90 deg; joints [76.189, -17.522, 83.89, 0, 23.632, 76.189]
  MoveL 4378 to (27.08, 67.5, -3.91) mm, rotated rx 180 ry 0 rz 90 deg; joints [76.24, -17.504, 83.888, 0, 23.616, 76.24]
  MoveL 4379 to (26.92, 69.01, -4.31) mm, rotated rx 180 ry 0 rz 90 deg; joints [76.288, -17.493, 83.912, 0, 23.581, 76.288]
  MoveL 4380 to (26.43, 70.45, -4.72) mm, rotated rx -180 ry 0 rz 90 deg; joints [76.331, -17.488, 83.959, 0, 23.53, 76.331]
  MoveL 4381 to (25.64, 71.74, -5.13) mm, rotated rx 180 ry 0 rz 90 deg; joints [76.366, -17.489, 84.025, 0, 23.464, 76.366]
  MoveL 4382 to (24.58, 72.83, -5.53) mm, rotated rx 180 ry 0 rz 90 deg; joints [76.394, -17.493, 84.107, 0, 23.386, 76.394]
  MoveL 4383 to (23.3, 73.66, -5.94) mm, rotated rx 180 ry 0 rz 90 deg; joints [76.411, -17.5, 84.199, 0, 23.301, 76.411]
  MoveL 4384 to (21.88, 74.18, -6.34) mm, rotated rx -180 ry 0 rz 90 deg; joints [76.416, -17.508, 84.297, 0, 23.212, 76.416]
  MoveL 4385 to (20.37, 74.35, -6.75) mm, rotated rx -180 ry 0 rz 90 deg; joints [76.41, -17.517, 84.394, 0, 23.122, 76.41]
  MoveL 4386 to (12.79, 74.48, -6.75) mm, rotated rx 180 ry 0 rz 90 deg; joints [76.354, -17.657, 84.939, 0, 22.718, 76.354]
  MoveL 4387 to (-27.79, 74.95, -6.75) mm, rotated rx -180 ry 0 rz 90 deg; joints [76.038, -18.362, 87.795, 0, 20.566, 76.038]
  MoveC 4388 to (-30.4, 71.63, -6.75) mm, rotated rx -180 ry 0 rz 90 deg; joints [75.905, -18.391, 87.918, 0, 20.473, 75.905] to (-29.95, 67.44, -6.75) mm, rotated rx 180 ry 0 rz 90 deg; joints [75.768, -18.366, 87.815, 0, 20.552, 75.768]
  MoveL 4389 to (-10.38, 55, -6.75) mm, rotated rx 180 ry 0 rz 90 deg; joints [75.521, -17.983, 86.232, 0, 21.751, 75.521]
  MoveC 4390 to (-8.85, 54.34, -6.75) mm, rotated rx -180 ry 0 rz 90 deg; joints [75.512, -17.953, 86.113, 0, 21.84, 75.512] to (-7.19, 54.2, -6.75) mm, rotated rx -180 ry 0 rz 90 deg; joints [75.521, -17.924, 85.994, 0, 21.93, 75.521]
  MoveC 4391 to (13.23, 55.7, -6.75) mm, rotated rx -180 ry 0 rz 90 deg; joints [75.743, -17.563, 84.575, 0, 22.989, 75.743] to (33.64, 57.24, -6.75) mm, rotated rx 180 ry 0 rz 90 deg; joints [75.96, -17.184, 83.132, 0, 24.051, 75.96]
  MoveC 4392 to (51.38, 58.85, -6.75) mm, rotated rx 180 ry 0 rz 90 deg; joints [76.153, -16.84, 81.864, 0, 24.976, 76.153] to (69.06, 60.95, -6.75) mm, rotated rx 180 ry 0 rz 90 deg; joints [76.358, -16.484, 80.588, 0, 25.896, 76.358]
  MoveC 4393 to (71.03, 62.01, -6.75) mm, rotated rx -180 ry 0 rz 90 deg; joints [76.407, -16.448, 80.46, 0, 25.988, 76.407] to (71.82, 64.1, -6.75) mm, rotated rx -180 ry 0 rz 90 deg; joints [76.479, -16.442, 80.438, 0, 26.003, 76.479]
  MoveL 4394 to (71.82, 69.65, -6.75) mm, rotated rx 180 ry 0 rz 90 deg; joints [76.656, -16.47, 80.538, 0, 25.932, 76.656]
  MoveC 4395 to (71.16, 71.4, -6.75) mm, rotated rx 180 ry 0 rz 90 deg; joints [76.706, -16.492, 80.618, 0, 25.874, 76.706] to (69.65, 72.49, -6.75) mm, rotated rx 180 ry 0 rz 90 deg; joints [76.73, -16.53, 80.751, 0, 25.779, 76.73]
  MoveL 4396 to (68.7, 72.6, -6.75) mm, rotated rx 180 ry 0 rz 90 deg; joints [76.726, -16.55, 80.824, 0, 25.727, 76.726]
  MoveL 4397 to (61.6, 72.99, -6.75) mm, rotated rx -180 ry 0 rz 90 deg; joints [76.685, -16.7, 81.36, 0, 25.34, 76.685]
  MoveC 4398 to (44.63, 73.76, -6.75) mm, rotated rx 180 ry 0 rz 90 deg; joints [76.58, -17.047, 82.626, 0, 24.422, 76.58] to (27.65, 74.22, -6.75) mm, rotated rx 180 ry 0 rz 90 deg; joints [76.463, -17.379, 83.868, 0, 23.511, 76.463]
  MoveL 4399 to (20.37, 74.35, -6.75) mm, rotated rx -180 ry 0 rz 90 deg; joints [76.41, -17.517, 84.394, 0, 23.122, 76.41]
  MoveL 4400 to (20.24, 66.8, -6.75) mm, rotated rx 180 ry 0 rz 90 deg; joints [76.162, -17.485, 84.272, 0, 23.213, 76.162]
  MoveL 4401 to (20.24, 66.8, -3.75) mm, rotated rx -180 ry 0 rz 90 deg; joints [76.162, -17.638, 84.373, 0, 23.265, 76.162]
  Establecer velocidad (1000.0 mm/s)
  MoveL 4402 to (20.24, 66.8, 10) mm, rotated rx -180 ry 0 rz 90 deg; joints [76.162, -18.34, 84.832, 0, 23.508, 76.162]
  Establecer velocidad (66.7 mm/s)
  MoveL 4403 to (36.53, 21.9, 10) mm, rotated rx -180 ry 0 rz 90 deg; joints [74.848, -17.795, 82.814, 0, 24.981, 74.848]
  MoveL 4404 to (36.53, 21.9, -3.5) mm, rotated rx 180 ry 0 rz 90 deg; joints [74.848, -17.111, 82.362, 0, 24.748, 74.848]
  MoveL 4405 to (36.68, 23.41, -3.91) mm, rotated rx 180 ry 0 rz 90 deg; joints [74.898, -17.095, 82.367, 0, 24.728, 74.898]
  MoveL 4406 to (36.46, 24.91, -4.31) mm, rotated rx 180 ry 0 rz 90 deg; joints [74.944, -17.087, 82.399, 0, 24.688, 74.944]
  MoveL 4407 to (35.92, 26.33, -4.72) mm, rotated rx -180 ry 0 rz 90 deg; joints [74.985, -17.085, 82.453, 0, 24.632, 74.985]
  MoveL 4408 to (35.07, 27.6, -5.13) mm, rotated rx 180 ry 0 rz 90 deg; joints [75.018, -17.088, 82.525, 0, 24.563, 75.018]
  MoveL 4409 to (33.97, 28.64, -5.53) mm, rotated rx -180 ry 0 rz 90 deg; joints [75.042, -17.094, 82.612, 0, 24.482, 75.042]
  MoveL 4410 to (32.67, 29.42, -5.94) mm, rotated rx 180 ry 0 rz 90 deg; joints [75.056, -17.104, 82.708, 0, 24.395, 75.056]
  MoveL 4411 to (31.22, 29.89, -6.34) mm, rotated rx -180 ry 0 rz 90 deg; joints [75.058, -17.114, 82.808, 0, 24.305, 75.058]
  MoveL 4412 to (29.71, 29.99, -6.75) mm, rotated rx -180 ry 0 rz 90 deg; joints [75.049, -17.123, 82.907, 0, 24.217, 75.049]
  MoveL 4413 to (9.95, 29.56, -6.75) mm, rotated rx -180 ry 0 rz 90 deg; joints [74.863, -17.497, 84.319, 0, 23.178, 74.863]
  MoveL 4414 to (9, 29.51, -6.75) mm, rotated rx 180 ry 0 rz 90 deg; joints [74.853, -17.514, 84.386, 0, 23.128, 74.853]
  MoveC 4415 to (6.46, 27.95, -6.75) mm, rotated rx 180 ry 0 rz 90 deg; joints [74.78, -17.553, 84.537, 0, 23.017, 74.78] to (5.55, 25.11, -6.75) mm, rotated rx 180 ry 0 rz 90 deg; joints [74.68, -17.556, 84.546, 0, 23.01, 74.68]
  MoveL 4416 to (5.62, 24.64, -6.75) mm, rotated rx -180 ry 0 rz 90 deg; joints [74.665, -17.552, 84.532, 0, 23.02, 74.665]
  MoveL 4417 to (5.79, 24.17, -6.75) mm, rotated rx 180 ry 0 rz 90 deg; joints [74.651, -17.547, 84.511, 0, 23.036, 74.651]
  MoveL 4418 to (10.96, 9.95, -6.75) mm, rotated rx 180 ry 0 rz 90 deg; joints [74.238, -17.377, 83.86, 0, 23.517, 74.238]
  MoveL 4419 to (11.27, 9.13, -6.75) mm, rotated rx -180 ry 0 rz 90 deg; joints [74.214, -17.367, 83.822, 0, 23.545, 74.214]
  MoveC 4420 to (11.76, 8.22, -6.75) mm, rotated rx 180 ry 0 rz 90 deg; joints [74.189, -17.353, 83.768, 0, 23.585, 74.189] to (12.48, 7.49, -6.75) mm, rotated rx -180 ry 0 rz 90 deg; joints [74.172, -17.335, 83.701, 0, 23.634, 74.172]
  MoveL 4421 to (28.29, -4.69, -6.75) mm, rotated rx -180 ry 0 rz 90 deg; joints [73.927, -16.962, 82.311, 0, 24.651, 73.927]
  MoveC 4422 to (30.11, -5.46, -6.75) mm, rotated rx 180 ry 0 rz 90 deg; joints [73.919, -16.921, 82.162, 0, 24.759, 73.919] to (32.08, -5.21, -6.75) mm, rotated rx 180 ry 0 rz 90 deg; joints [73.945, -16.884, 82.024, 0, 24.859, 73.945]
  MoveC 4423 to (33.25, -4.65, -6.75) mm, rotated rx 180 ry 0 rz 90 deg; joints [73.974, -16.864, 81.951, 0, 24.913, 73.974] to (34.17, -3.74, -6.75) mm, rotated rx -180 ry 0 rz 90 deg; joints [74.011, -16.85, 81.903, 0, 24.947, 74.011]
  MoveL 4424 to (37.85, 1.42, -6.75) mm, rotated rx -180 ry 0 rz 90 deg; joints [74.208, -16.806, 81.741, 0, 25.065, 74.208]
  MoveL 4425 to (53.01, 22.74, -6.75) mm, rotated rx -180 ry 0 rz 90 deg; joints [75.016, -16.616, 81.058, 0, 25.558, 75.016]
  MoveL 4426 to (53.54, 23.52, -6.75) mm, rotated rx -180 ry 0 rz 90 deg; joints [75.045, -16.609, 81.033, 0, 25.576, 75.045]
  MoveC 4427 to (53.22, 27.52, -6.75) mm, rotated rx -180 ry 0 rz 90 deg; joints [75.169, -16.638, 81.136, 0, 25.502, 75.169] to (50.41, 30.4, -6.75) mm, rotated rx 180 ry 0 rz 90 deg; joints [75.237, -16.711, 81.4, 0, 25.312, 75.237]
  MoveL 4428 to (45.96, 30.35, -6.75) mm, rotated rx 180 ry 0 rz 90 deg; joints [75.198, -16.802, 81.727, 0, 25.075, 75.198]
  MoveL 4429 to (29.71, 29.99, -6.75) mm, rotated rx -180 ry 0 rz 90 deg; joints [75.049, -17.123, 82.907, 0, 24.217, 75.049]
  MoveL 4430 to (29.87, 22.45, -6.75) mm, rotated rx 180 ry 0 rz 90 deg; joints [74.808, -17.08, 82.747, 0, 24.333, 74.808]
  MoveL 4431 to (29.87, 22.45, -3.75) mm, rotated rx 180 ry 0 rz 90 deg; joints [74.808, -17.233, 82.849, 0, 24.384, 74.808]
  Establecer velocidad (1000.0 mm/s)
  MoveL 4432 to (29.87, 22.45, 10) mm, rotated rx -180 ry 0 rz 90 deg; joints [74.808, -17.931, 83.309, 0, 24.622, 74.808]
  Establecer velocidad (66.7 mm/s)
  MoveL 4433 to (64.5, -32.45, 10) mm, rotated rx 180 ry 0 rz 90 deg; joints [73.389, -16.878, 79.601, 0, 27.278, 73.389]
  MoveL 4434 to (64.5, -32.45, -3.5) mm, rotated rx 180 ry 0 rz 90 deg; joints [73.389, -16.202, 79.146, 0, 27.055, 73.389]
  MoveL 4435 to (66.01, -32.63, -3.91) mm, rotated rx 180 ry 0 rz 90 deg; joints [73.397, -16.147, 79.015, 0, 27.132, 73.397]
  MoveL 4436 to (67.52, -32.45, -4.31) mm, rotated rx 180 ry 0 rz 90 deg; joints [73.417, -16.095, 78.892, 0, 27.203, 73.417]
  MoveL 4437 to (68.95, -31.94, -4.72) mm, rotated rx 180 ry 0 rz 90 deg; joints [73.446, -16.046, 78.782, 0, 27.265, 73.446]
  MoveL 4438 to (70.23, -31.12, -5.13) mm, rotated rx 180 ry 0 rz 90 deg; joints [73.483, -16.003, 78.689, 0, 27.314, 73.483]
  MoveL 4439 to (71.3, -30.04, -5.53) mm, rotated rx 180 ry 0 rz 90 deg; joints [73.526, -15.966, 78.619, 0, 27.347, 73.526]
  MoveL 4440 to (72.1, -28.76, -5.94) mm, rotated rx 180 ry 0 rz 90 deg; joints [73.573, -15.936, 78.573, 0, 27.363, 73.573]
  MoveL 4441 to (72.6, -27.32, -6.34) mm, rotated rx 180 ry 0 rz 90 deg; joints [73.622, -15.914, 78.553, 0, 27.361, 73.622]
  MoveL 4442 to (72.74, -25.81, -6.75) mm, rotated rx 180 ry 0 rz 90 deg; joints [73.67, -15.901, 78.562, 0, 27.338, 73.67]
  MoveL 4443 to (72.74, -12.45, -6.75) mm, rotated rx -180 ry 0 rz 90 deg; joints [74.084, -15.986, 78.854, 0, 27.132, 74.084]
  MoveC 4444 to (70.41, -9.39, -6.75) mm, rotated rx -180 ry 0 rz 90 deg; joints [74.158, -16.057, 79.096, 0, 26.96, 74.158] to (66.81, -8.02, -6.75) mm, rotated rx 180 ry 0 rz 90 deg; joints [74.169, -16.143, 79.396, 0, 26.747, 74.169]
  MoveL 4445 to (65.46, -8.23, -6.75) mm, rotated rx 180 ry 0 rz 90 deg; joints [74.151, -16.171, 79.493, 0, 26.678, 74.151]
  MoveL 4446 to (54.19, -23.59, -6.75) mm, rotated rx 180 ry 0 rz 90 deg; joints [73.57, -16.318, 80.003, 0, 26.315, 73.57]
  MoveC 4447 to (53.6, -24.76, -6.75) mm, rotated rx -180 ry 0 rz 90 deg; joints [73.528, -16.323, 80.022, 0, 26.302, 73.528] to (53.4, -26.06, -6.75) mm, rotated rx 180 ry 0 rz 90 deg; joints [73.485, -16.319, 80.008, 0, 26.312, 73.485]
  MoveC 4448 to (53.63, -27.27, -6.75) mm, rotated rx 180 ry 0 rz 90 deg; joints [73.449, -16.306, 79.964, 0, 26.343, 73.449] to (54.27, -28.32, -6.75) mm, rotated rx 180 ry 0 rz 90 deg; joints [73.423, -16.286, 79.893, 0, 26.394, 73.423]
  MoveL 4449 to (56.46, -30.8, -6.75) mm, rotated rx 180 ry 0 rz 90 deg; joints [73.366, -16.224, 79.675, 0, 26.549, 73.366]
  MoveL 4450 to (65.86, -41.37, -6.75) mm, rotated rx 180 ry 0 rz 90 deg; joints [73.126, -15.95, 78.732, 0, 27.219, 73.126]
  MoveL 4451 to (65.9, -41.39, -6.75) mm, rotated rx 180 ry 0 rz 90 deg; joints [73.126, -15.949, 78.728, 0, 27.221, 73.126]
  MoveC 4452 to (69.21, -41.05, -6.75) mm, rotated rx 180 ry 0 rz 90 deg; joints [73.167, -15.878, 78.486, 0, 27.392, 73.167] to (71.74, -38.89, -6.75) mm, rotated rx -180 ry 0 rz 90 deg; joints [73.257, -15.836, 78.344, 0, 27.492, 73.257]
  MoveL 4453 to (72.65, -37.43, -6.75) mm, rotated rx -180 ry 0 rz 90 deg; joints [73.311, -15.826, 78.308, 0, 27.518, 73.311]
  MoveL 4454 to (72.74, -37.21, -6.75) mm, rotated rx 180 ry 0 rz 90 deg; joints [73.318, -15.825, 78.307, 0, 27.519, 73.318]
  MoveL 4455 to (72.74, -25.81, -6.75) mm, rotated rx 180 ry 0 rz 90 deg; joints [73.67, -15.901, 78.562, 0, 27.338, 73.67]
  MoveL 4456 to (65.19, -25.81, -6.75) mm, rotated rx -180 ry 0 rz 90 deg; joints [73.601, -16.067, 79.132, 0, 26.935, 73.601]
  MoveL 4457 to (65.19, -25.81, -3.75) mm, rotated rx 180 ry 0 rz 90 deg; joints [73.601, -16.217, 79.234, 0, 26.983, 73.601]
  Establecer velocidad (1000.0 mm/s)
  MoveL 4458 to (65.19, -25.81, 10) mm, rotated rx 180 ry 0 rz 90 deg; joints [73.601, -16.907, 79.697, 0, 27.21, 73.601]
  Establecer velocidad (66.7 mm/s)
  MoveL 4459 to (16.69, -66.38, 10) mm, rotated rx -180 ry 0 rz 90 deg; joints [71.866, -17.663, 82.339, 0, 25.324, 71.866]
  MoveL 4460 to (16.69, -66.38, -3.5) mm, rotated rx 180 ry 0 rz 90 deg; joints [71.866, -16.98, 81.887, 0, 25.093, 71.866]
  MoveL 4461 to (16.52, -67.88, -3.91) mm, rotated rx -180 ry 0 rz 90 deg; joints [71.817, -16.953, 81.849, 0, 25.104, 71.817]
  MoveL 4462 to (16.73, -69.39, -4.31) mm, rotated rx 180 ry 0 rz 90 deg; joints [71.772, -16.918, 81.785, 0, 25.134, 71.772]
  MoveL 4463 to (17.26, -70.81, -4.72) mm, rotated rx 180 ry 0 rz 90 deg; joints [71.733, -16.878, 81.699, 0, 25.179, 71.733]
  MoveL 4464 to (18.1, -72.08, -5.13) mm, rotated rx 180 ry 0 rz 90 deg; joints [71.702, -16.832, 81.594, 0, 25.238, 71.702]
  MoveL 4465 to (19.19, -73.13, -5.53) mm, rotated rx 180 ry 0 rz 90 deg; joints [71.681, -16.782, 81.476, 0, 25.307, 71.681]
  MoveL 4466 to (20.49, -73.92, -5.94) mm, rotated rx 180 ry 0 rz 90 deg; joints [71.67, -16.73, 81.349, 0, 25.382, 71.67]
  MoveL 4467 to (21.94, -74.4, -6.34) mm, rotated rx 180 ry 0 rz 90 deg; joints [71.67, -16.678, 81.219, 0, 25.459, 71.67]
  MoveL 4468 to (23.45, -74.51, -6.75) mm, rotated rx -180 ry 0 rz 90 deg; joints [71.682, -16.626, 81.092, 0, 25.533, 71.682]
  MoveC 4469 to (36.36, -74.3, -6.75) mm, rotated rx -180 ry 0 rz 90 deg; joints [71.82, -16.361, 80.153, 0, 26.207, 71.82] to (49.26, -74.06, -6.75) mm, rotated rx 180 ry 0 rz 90 deg; joints [71.958, -16.088, 79.205, 0, 26.883, 71.958]
  MoveC 4470 to (51.34, -72.24, -6.75) mm, rotated rx -180 ry 0 rz 90 deg; joints [72.035, -16.056, 79.094, 0, 26.962, 72.035] to (52.29, -69.65, -6.75) mm, rotated rx 180 ry 0 rz 90 deg; joints [72.124, -16.053, 79.085, 0, 26.968, 72.124]
  MoveC 4471 to (52.36, -67.86, -6.75) mm, rotated rx -180 ry 0 rz 90 deg; joints [72.18, -16.064, 79.123, 0, 26.941, 72.18] to (51.57, -66.25, -6.75) mm, rotated rx -180 ry 0 rz 90 deg; joints [72.221, -16.093, 79.221, 0, 26.872, 72.221]
  MoveL 4472 to (49.64, -63.97, -6.75) mm, rotated rx 180 ry 0 rz 90 deg; joints [72.273, -16.15, 79.419, 0, 26.731, 72.273]
  MoveL 4473 to (26.05, -36.45, -6.75) mm, rotated rx 180 ry 0 rz 90 deg; joints [72.9, -16.818, 81.786, 0, 25.032, 72.9]
  MoveC 4474 to (25.72, -36.09, -6.75) mm, rotated rx 180 ry 0 rz 90 deg; joints [72.908, -16.827, 81.819, 0, 25.008, 72.908] to (25.35, -35.76, -6.75) mm, rotated rx 180 ry 0 rz 90 deg; joints [72.915, -16.837, 81.853, 0, 24.984, 72.915]
  MoveL 4475 to (11.85, -24.95, -6.75) mm, rotated rx 180 ry 0 rz 90 deg; joints [73.127, -17.166, 83.065, 0, 24.101, 73.127]
  MoveC 4476 to (9.63, -24.46, -6.75) mm, rotated rx 180 ry 0 rz 90 deg; joints [73.122, -17.211, 83.234, 0, 23.977, 73.122] to (7.46, -25.11, -6.75) mm, rotated rx -180 ry 0 rz 90 deg; joints [73.079, -17.249, 83.375, 0, 23.873, 73.079]
  MoveL 4477 to (7.24, -25.24, -6.75) mm, rotated rx -180 ry 0 rz 90 deg; joints [73.073, -17.252, 83.389, 0, 23.864, 73.073]
  MoveC 4478 to (6.35, -26.01, -6.75) mm, rotated rx 180 ry 0 rz 90 deg; joints [73.04, -17.265, 83.435, 0, 23.829, 73.04] to (5.83, -27.06, -6.75) mm, rotated rx -180 ry 0 rz 90 deg; joints [73.001, -17.268, 83.449, 0, 23.819, 73.001]
  MoveL 4479 to (-5.53, -69.65, -6.75) mm, rotated rx -180 ry 0 rz 90 deg; joints [71.532, -17.226, 83.289, 0, 23.937, 71.532]
  MoveC 4480 to (-5.1, -72.93, -6.75) mm, rotated rx 180 ry 0 rz 90 deg; joints [71.432, -17.197, 83.18, 0, 24.016, 71.432] to (-2.37, -74.81, -6.75) mm, rotated rx 180 ry 0 rz 90 deg; joints [71.402, -17.133, 82.942, 0, 24.191, 71.402]
  MoveL 4481 to (-1.42, -74.83, -6.75) mm, rotated rx 180 ry 0 rz 90 deg; joints [71.412, -17.114, 82.874, 0, 24.241, 71.412]
  MoveC 4482 to (11.01, -74.69, -6.75) mm, rotated rx 180 ry 0 rz 90 deg; joints [71.547, -16.874, 81.987, 0, 24.886, 71.547] to (23.45, -74.51, -6.75) mm, rotated rx -180 ry 0 rz 90 deg; joints [71.682, -16.626, 81.092, 0, 25.533, 71.682]
  MoveL 4483 to (23.33, -66.96, -6.75) mm, rotated rx 180 ry 0 rz 90 deg; joints [71.916, -16.678, 81.281, 0, 25.397, 71.916]
  MoveL 4484 to (23.33, -66.96, -3.75) mm, rotated rx 180 ry 0 rz 90 deg; joints [71.916, -16.83, 81.383, 0, 25.447, 71.916]
  Establecer velocidad (1000.0 mm/s)
  MoveL 4485 to (23.33, -66.96, 10) mm, rotated rx -180 ry 0 rz 90 deg; joints [71.916, -17.524, 81.844, 0, 25.681, 71.916]
  Establecer velocidad (66.7 mm/s)
  MoveL 4486 to (-34.48, -50.84, 10) mm, rotated rx 180 ry 0 rz 90 deg; joints [71.827, -18.724, 86.311, 0, 22.413, 71.827]
  MoveL 4487 to (-34.48, -50.84, -3.5) mm, rotated rx -180 ry 0 rz 90 deg; joints [71.827, -18.03, 85.861, 0, 22.169, 71.827]
  MoveL 4488 to (-33.07, -51.39, -3.91) mm, rotated rx 180 ry 0 rz 90 deg; joints [71.824, -17.982, 85.737, 0, 22.244, 71.824]
  MoveL 4489 to (-31.57, -51.6, -4.31) mm, rotated rx -180 ry 0 rz 90 deg; joints [71.833, -17.933, 85.615, 0, 22.318, 71.833]
  MoveL 4490 to (-30.05, -51.46, -4.72) mm, rotated rx 180 ry 0 rz 90 deg; joints [71.853, -17.887, 85.499, 0, 22.387, 71.853]
  MoveL 4491 to (-28.61, -51, -5.13) mm, rotated rx 180 ry 0 rz 90 deg; joints [71.884, -17.843, 85.396, 0, 22.447, 71.884]
  MoveL 4492 to (-27.3, -50.22, -5.53) mm, rotated rx -180 ry 0 rz 90 deg; joints [71.923, -17.803, 85.309, 0, 22.495, 71.923]
  MoveL 4493 to (-26.2, -49.18, -5.94) mm, rotated rx 180 ry 0 rz 90 deg; joints [71.968, -17.769, 85.242, 0, 22.527, 71.968]
  MoveL 4494 to (-25.35, -47.91, -6.34) mm, rotated rx 180 ry 0 rz 90 deg; joints [72.017, -17.74, 85.198, 0, 22.543, 72.017]
  MoveL 4495 to (-24.84, -46.49, -6.75) mm, rotated rx -180 ry 0 rz 90 deg; joints [72.069, -17.719, 85.181, 0, 22.538, 72.069]
  MoveL 4496 to (-18.88, -23.63, -6.75) mm, rotated rx 180 ry 0 rz 90 deg; joints [72.868, -17.741, 85.269, 0, 22.472, 72.868]
  MoveC 4497 to (-18.7, -22.76, -6.75) mm, rotated rx 180 ry 0 rz 90 deg; joints [72.898, -17.743, 85.275, 0, 22.468, 72.898] to (-18.59, -21.88, -6.75) mm, rotated rx 180 ry 0 rz 90 deg; joints [72.927, -17.746, 85.286, 0, 22.46, 72.927]
  MoveC 4498 to (-19.42, -19.61, -6.75) mm, rotated rx 180 ry 0 rz 90 deg; joints [72.993, -17.773, 85.393, 0, 22.38, 72.993] to (-21.34, -18.14, -6.75) mm, rotated rx -180 ry 0 rz 90 deg; joints [73.021, -17.815, 85.558, 0, 22.256, 73.021]
  MoveC 4499 to (-22.27, -17.92, -6.75) mm, rotated rx 180 ry 0 rz 90 deg; joints [73.019, -17.832, 85.627, 0, 22.205, 73.019] to (-23.21, -17.99, -6.75) mm, rotated rx -180 ry 0 rz 90 deg; joints [73.008, -17.848, 85.692, 0, 22.156, 73.008]
  MoveL 4500 to (-72.29, -28.43, -6.75) mm, rotated rx -180 ry 0 rz 90 deg; joints [72.158, -18.601, 88.82, 0, 19.78, 72.158]
  MoveC 4501 to (-73.82, -29.09, -6.75) mm, rotated rx -180 ry 0 rz 90 deg; joints [72.12, -18.621, 88.909, 0, 19.712, 72.12] to (-75, -30.29, -6.75) mm, rotated rx 180 ry 0 rz 90 deg; joints [72.068, -18.633, 88.961, 0, 19.671, 72.068]
  MoveC 4502 to (-75.42, -31.33, -6.75) mm, rotated rx 180 ry 0 rz 90 deg; joints [72.028, -18.634, 88.967, 0, 19.667, 72.028] to (-75.56, -32.45, -6.75) mm, rotated rx 180 ry 0 rz 90 deg; joints [71.99, -18.631, 88.952, 0, 19.679, 71.99]
  MoveL 4503 to (-75.56, -70.6, -6.75) mm, rotated rx 180 ry 0 rz 90 deg; joints [70.731, -18.431, 88.091, 0, 20.341, 70.731]
  MoveL 4504 to (-75.52, -71.27, -6.75) mm, rotated rx 180 ry 0 rz 90 deg; joints [70.709, -18.427, 88.072, 0, 20.355, 70.709]
  MoveC 4505 to (-74.52, -73.63, -6.75) mm, rotated rx 180 ry 0 rz 90 deg; joints [70.644, -18.398, 87.95, 0, 20.448, 70.644] to (-72.26, -74.82, -6.75) mm, rotated rx -180 ry 0 rz 90 deg; joints [70.631, -18.356, 87.77, 0, 20.586, 70.631]
  MoveL 4506 to (-71.55, -74.92, -6.75) mm, rotated rx -180 ry 0 rz 90 deg; joints [70.636, -18.344, 87.72, 0, 20.624, 70.636]
  MoveL 4507 to (-35.26, -74.64, -6.75) mm, rotated rx -180 ry 0 rz 90 deg; joints [71.052, -17.737, 85.252, 0, 22.485, 71.052]
  MoveC 4508 to (-33.23, -74.06, -6.75) mm, rotated rx 180 ry 0 rz 90 deg; joints [71.093, -17.705, 85.126, 0, 22.579, 71.093] to (-31.8, -72.51, -6.75) mm, rotated rx -180 ry 0 rz 90 deg; joints [71.158, -17.689, 85.063, 0, 22.626, 71.158]
  MoveC 4509 to (-31.48, -71.8, -6.75) mm, rotated rx -180 ry 0 rz 90 deg; joints [71.185, -17.687, 85.058, 0, 22.63, 71.185] to (-31.24, -71.06, -6.75) mm, rotated rx 180 ry 0 rz 90 deg; joints [71.211, -17.688, 85.059, 0, 22.629, 71.211]
  MoveL 4510 to (-24.84, -46.49, -6.75) mm, rotated rx -180 ry 0 rz 90 deg; joints [72.069, -17.719, 85.181, 0, 22.538, 72.069]
  MoveL 4511 to (-32.14, -44.58, -6.75) mm, rotated rx 180 ry 0 rz 90 deg; joints [72.054, -17.858, 85.731, 0, 22.127, 72.054]
  MoveL 4512 to (-32.14, -44.58, -3.75) mm, rotated rx -180 ry 0 rz 90 deg; joints [72.054, -18.012, 85.832, 0, 22.18, 72.054]
  Establecer velocidad (1000.0 mm/s)
  MoveL 4513 to (-32.14, -44.58, 10) mm, rotated rx -180 ry 0 rz 90 deg; joints [72.054, -18.719, 86.291, 0, 22.428, 72.054]
  Establecer velocidad (66.7 mm/s)
  MoveL 4514 to (-67.32, 36.29, 10) mm, rotated rx -180 ry 0 rz 90 deg; joints [74.382, -19.697, 90.352, 0, 19.344, 74.382]
  MoveL 4515 to (-67.32, 36.29, -3.5) mm, rotated rx -180 ry 0 rz 90 deg; joints [74.382, -18.99, 89.902, 0, 19.088, 74.382]
  MoveL 4516 to (-68.82, 36.47, -3.91) mm, rotated rx 180 ry 0 rz 90 deg; joints [74.374, -18.992, 89.993, 0, 18.999, 74.374]
  MoveL 4517 to (-70.33, 36.29, -4.31) mm, rotated rx 180 ry 0 rz 90 deg; joints [74.353, -18.992, 90.077, 0, 18.916, 74.353]
  MoveL 4518 to (-71.76, 35.78, -4.72) mm, rotated rx -180 ry 0 rz 90 deg; joints [74.322, -18.99, 90.149, 0, 18.841, 74.322]
  MoveL 4519 to (-73.05, 34.96, -5.13) mm, rotated rx -180 ry 0 rz 90 deg; joints [74.282, -18.984, 90.206, 0, 18.778, 74.282]
  MoveL 4520 to (-74.11, 33.88, -5.53) mm, rotated rx -180 ry 0 rz 90 deg; joints [74.235, -18.974, 90.243, 0, 18.731, 74.235]
  MoveL 4521 to (-74.92, 32.6, -5.94) mm, rotated rx 180 ry 0 rz 90 deg; joints [74.184, -18.959, 90.259, 0, 18.7, 74.184]
  MoveL 4522 to (-75.42, 31.16, -6.34) mm, rotated rx -180 ry 0 rz 90 deg; joints [74.13, -18.939, 90.251, 0, 18.688, 74.13]
  MoveL 4523 to (-75.56, 29.65, -6.75) mm, rotated rx -180 ry 0 rz 90 deg; joints [74.077, -18.914, 90.218, 0, 18.696, 74.077]
  MoveL 4524 to (-75.56, 1.42, -6.75) mm, rotated rx 180 ry 0 rz 90 deg; joints [73.123, -18.791, 89.663, 0, 19.128, 73.123]
  MoveL 4525 to (-75.55, 0.47, -6.75) mm, rotated rx -180 ry 0 rz 90 deg; joints [73.091, -18.787, 89.643, 0, 19.143, 73.091]
  MoveC 4526 to (-74.37, -2.28, -6.75) mm, rotated rx -180 ry 0 rz 90 deg; joints [73.01, -18.757, 89.509, 0, 19.248, 73.01] to (-71.57, -3.34, -6.75) mm, rotated rx 180 ry 0 rz 90 deg; joints [73.003, -18.71, 89.299, 0, 19.41, 73.003]
  MoveC 4527 to (-70.81, -3.27, -6.75) mm, rotated rx -180 ry 0 rz 90 deg; joints [73.013, -18.698, 89.25, 0, 19.448, 73.013] to (-70.06, -3.15, -6.75) mm, rotated rx -180 ry 0 rz 90 deg; joints [73.025, -18.688, 89.202, 0, 19.485, 73.025]
  MoveL 4528 to (-68.7, -2.86, -6.75) mm, rotated rx -180 ry 0 rz 90 deg; joints [73.049, -18.668, 89.117, 0, 19.551, 73.049]
  MoveL 4529 to (-22.27, 7.83, -6.75) mm, rotated rx 180 ry 0 rz 90 deg; joints [73.86, -17.965, 86.161, 0, 21.804, 73.86]
  MoveL 4530 to (-20.53, 8.25, -6.75) mm, rotated rx -180 ry 0 rz 90 deg; joints [73.89, -17.937, 86.048, 0, 21.889, 73.89]
  MoveC 4531 to (-19.8, 8.52, -6.75) mm, rotated rx 180 ry 0 rz 90 deg; joints [73.906, -17.926, 86.003, 0, 21.923, 73.906] to (-19.14, 8.94, -6.75) mm, rotated rx 180 ry 0 rz 90 deg; joints [73.926, -17.917, 85.965, 0, 21.951, 73.926]
  MoveC 4532 to (-17.85, 10.83, -6.75) mm, rotated rx -180 ry 0 rz 90 deg; joints [74, -17.904, 85.913, 0, 21.991, 74] to (-17.82, 13.12, -6.75) mm, rotated rx -180 ry 0 rz 90 deg; joints [74.075, -17.915, 85.957, 0, 21.958, 74.075]
  MoveL 4533 to (-18, 13.74, -6.75) mm, rotated rx -180 ry 0 rz 90 deg; joints [74.094, -17.921, 85.982, 0, 21.939, 74.094]
  MoveL 4534 to (-24.72, 32.46, -6.75) mm, rotated rx 180 ry 0 rz 90 deg; joints [74.649, -18.126, 86.813, 0, 21.312, 74.649]
  MoveC 4535 to (-25.42, 33.72, -6.75) mm, rotated rx 180 ry 0 rz 90 deg; joints [74.684, -18.143, 86.886, 0, 21.258, 74.684] to (-26.49, 34.68, -6.75) mm, rotated rx 180 ry 0 rz 90 deg; joints [74.706, -18.166, 86.978, 0, 21.188, 74.706]
  MoveL 4536 to (-68.7, 61.75, -6.75) mm, rotated rx -180 ry 0 rz 90 deg; joints [75.236, -18.942, 90.349, 0, 18.593, 75.236]
  MoveC 4537 to (-69.84, 62.36, -6.75) mm, rotated rx 180 ry 0 rz 90 deg; joints [75.247, -18.961, 90.435, 0, 18.526, 75.247] to (-71.07, 62.76, -6.75) mm, rotated rx -180 ry 0 rz 90 deg; joints [75.249, -18.98, 90.524, 0, 18.456, 75.249]
  MoveC 4538 to (-73.65, 62.18, -6.75) mm, rotated rx -180 ry 0 rz 90 deg; joints [75.206, -19.015, 90.687, 0, 18.329, 75.206] to (-75.37, 60.18, -6.75) mm, rotated rx 180 ry 0 rz 90 deg; joints [75.122, -19.032, 90.766, 0, 18.266, 75.122]
  MoveC 4539 to (-75.51, 59.51, -6.75) mm, rotated rx -180 ry 0 rz 90 deg; joints [75.097, -19.032, 90.764, 0, 18.268, 75.097] to (-75.56, 58.82, -6.75) mm, rotated rx 180 ry 0 rz 90 deg; joints [75.073, -19.03, 90.755, 0, 18.275, 75.073]
  MoveL 4540 to (-75.56, 29.65, -6.75) mm, rotated rx -180 ry 0 rz 90 deg; joints [74.077, -18.914, 90.218, 0, 18.696, 74.077]
  MoveL 4541 to (-68.01, 29.65, -6.75) mm, rotated rx -180 ry 0 rz 90 deg; joints [74.15, -18.802, 89.713, 0, 19.089, 74.15]
  MoveL 4542 to (-68.01, 29.65, -3.75) mm, rotated rx -180 ry 0 rz 90 deg; joints [74.15, -18.959, 89.814, 0, 19.145, 74.15]
  Establecer velocidad (1000.0 mm/s)
  MoveL 4543 to (-68.01, 29.65, 10) mm, rotated rx 180 ry 0 rz 90 deg; joints [74.15, -19.679, 90.273, 0, 19.406, 74.15]
  Establecer velocidad (66.7 mm/s)
  MoveL 4544 to (-67.11, 36.29, 10) mm, rotated rx -180 ry 0 rz 90 deg; joints [74.384, -19.693, 90.338, 0, 19.355, 74.384]
  MoveL 4545 to (-67.11, 36.29, -3.75) mm, rotated rx 180 ry 0 rz 90 deg; joints [74.384, -18.974, 89.88, 0, 19.094, 74.384]
  MoveL 4546 to (-68.62, 36.47, -4.16) mm, rotated rx 180 ry 0 rz 90 deg; joints [74.376, -18.976, 89.97, 0, 19.005, 74.376]
  MoveL 4547 to (-70.13, 36.29, -4.56) mm, rotated rx 180 ry 0 rz 90 deg; joints [74.355, -18.976, 90.054, 0, 18.922, 74.355]
  MoveL 4548 to (-71.56, 35.78, -4.97) mm, rotated rx -180 ry 0 rz 90 deg; joints [74.324, -18.974, 90.127, 0, 18.847, 74.324]
  MoveL 4549 to (-72.84, 34.96, -5.37) mm, rotated rx 180 ry 0 rz 90 deg; joints [74.284, -18.968, 90.183, 0, 18.785, 74.284]
  MoveL 4550 to (-73.91, 33.88, -5.78) mm, rotated rx 180 ry 0 rz 90 deg; joints [74.237, -18.958, 90.221, 0, 18.737, 74.237]
  MoveL 4551 to (-74.71, 32.6, -6.19) mm, rotated rx -180 ry 0 rz 90 deg; joints [74.185, -18.943, 90.237, 0, 18.706, 74.185]
  MoveL 4552 to (-75.21, 31.16, -6.59) mm, rotated rx 180 ry 0 rz 90 deg; joints [74.132, -18.923, 90.229, 0, 18.694, 74.132]
  MoveL 4553 to (-75.35, 29.65, -7) mm, rotated rx 180 ry 0 rz 90 deg; joints [74.079, -18.897, 90.196, 0, 18.702, 74.079]
  MoveL 4554 to (-75.35, 1.42, -7) mm, rotated rx -180 ry 0 rz 90 deg; joints [73.125, -18.775, 89.641, 0, 19.134, 73.125]
  MoveL 4555 to (-75.34, 0.5, -7) mm, rotated rx -180 ry 0 rz 90 deg; joints [73.094, -18.771, 89.622, 0, 19.149, 73.094]
  MoveC 4556 to (-74.28, -2.05, -7) mm, rotated rx -180 ry 0 rz 90 deg; joints [73.019, -18.743, 89.499, 0, 19.244, 73.019] to (-71.76, -3.14, -7) mm, rotated rx 180 ry 0 rz 90 deg; joints [73.008, -18.7, 89.308, 0, 19.393, 73.008]
  MoveC 4557 to (-71.03, -3.12, -7) mm, rotated rx 180 ry 0 rz 90 deg; joints [73.016, -18.689, 89.259, 0, 19.43, 73.016] to (-70.31, -3.01, -7) mm, rotated rx 180 ry 0 rz 90 deg; joints [73.027, -18.679, 89.214, 0, 19.465, 73.027]
  MoveL 4558 to (-66.81, -2.22, -7) mm, rotated rx 180 ry 0 rz 90 deg; joints [73.089, -18.629, 88.995, 0, 19.635, 73.089]
  MoveL 4559 to (-27.01, 6.94, -7) mm, rotated rx 180 ry 0 rz 90 deg; joints [73.786, -18.029, 86.463, 0, 21.566, 73.786]
  MoveL 4560 to (-20.83, 8.36, -7) mm, rotated rx 180 ry 0 rz 90 deg; joints [73.891, -17.93, 86.063, 0, 21.867, 73.891]
  MoveC 4561 to (-18.39, 10.16, -7) mm, rotated rx -180 ry 0 rz 90 deg; joints [73.973, -17.897, 85.929, 0, 21.968, 73.973] to (-18.04, 13.18, -7) mm, rotated rx -180 ry 0 rz 90 deg; joints [74.075, -17.906, 85.965, 0, 21.941, 74.075]
  MoveL 4562 to (-18.21, 13.74, -7) mm, rotated rx -180 ry 0 rz 90 deg; joints [74.092, -17.911, 85.988, 0, 21.924, 74.092]
  MoveL 4563 to (-24.84, 32.29, -7) mm, rotated rx -180 ry 0 rz 90 deg; joints [74.642, -18.114, 86.81, 0, 21.304, 74.642]
  MoveC 4564 to (-25.55, 33.56, -7) mm, rotated rx 180 ry 0 rz 90 deg; joints [74.678, -18.132, 86.883, 0, 21.249, 74.678] to (-26.62, 34.53, -7) mm, rotated rx 180 ry 0 rz 90 deg; joints [74.7, -18.154, 86.976, 0, 21.178, 74.7]
  MoveL 4565 to (-68.7, 61.53, -7) mm, rotated rx 180 ry 0 rz 90 deg; joints [75.228, -18.928, 90.336, 0, 18.592, 75.228]
  MoveC 4566 to (-69.62, 62.04, -7) mm, rotated rx -180 ry 0 rz 90 deg; joints [75.238, -18.943, 90.407, 0, 18.537, 75.238] to (-70.6, 62.44, -7) mm, rotated rx 180 ry 0 rz 90 deg; joints [75.242, -18.959, 90.479, 0, 18.48, 75.242]
  MoveC 4567 to (-73.46, 61.97, -7) mm, rotated rx 180 ry 0 rz 90 deg; joints [75.201, -18.999, 90.662, 0, 18.337, 75.201] to (-75.27, 59.72, -7) mm, rotated rx 180 ry 0 rz 90 deg; joints [75.107, -19.016, 90.743, 0, 18.273, 75.107]
  MoveC 4568 to (-75.34, 59, -7) mm, rotated rx 180 ry 0 rz 90 deg; joints [75.082, -19.014, 90.735, 0, 18.279, 75.082] to (-75.35, 58.28, -7) mm, rotated rx 180 ry 0 rz 90 deg; joints [75.057, -19.012, 90.723, 0, 18.289, 75.057]
  MoveL 4569 to (-75.35, 29.65, -7) mm, rotated rx 180 ry 0 rz 90 deg; joints [74.079, -18.897, 90.196, 0, 18.702, 74.079]
  MoveL 4570 to (-67.8, 29.65, -7) mm, rotated rx 180 ry 0 rz 90 deg; joints [74.152, -18.786, 89.691, 0, 19.095, 74.152]
  MoveL 4571 to (-67.8, 29.65, -4) mm, rotated rx 180 ry 0 rz 90 deg; joints [74.152, -18.943, 89.792, 0, 19.151, 74.152]
  Establecer velocidad (1000.0 mm/s)
  MoveL 4572 to (-67.8, 29.65, 10) mm, rotated rx -180 ry 0 rz 90 deg; joints [74.152, -19.676, 90.259, 0, 19.416, 74.152]
  Establecer velocidad (66.7 mm/s)
  MoveL 4573 to (-39.4, -30.05, 10) mm, rotated rx -180 ry 0 rz 90 deg; joints [72.451, -18.926, 87.112, 0, 21.814, 72.451]
  MoveL 4574 to (-39.4, -30.05, -3.75) mm, rotated rx 180 ry 0 rz 90 deg; joints [72.451, -18.217, 86.654, 0, 21.563, 72.451]
  MoveL 4575 to (-39.53, -28.53, -4.16) mm, rotated rx 180 ry 0 rz 90 deg; joints [72.499, -18.206, 86.682, 0, 21.524, 72.499]
  MoveL 4576 to (-40.02, -27.1, -4.56) mm, rotated rx -180 ry 0 rz 90 deg; joints [72.541, -18.201, 86.733, 0, 21.468, 72.541]
  MoveL 4577 to (-40.82, -25.8, -4.97) mm, rotated rx -180 ry 0 rz 90 deg; joints [72.575, -18.2, 86.802, 0, 21.398, 72.575]
  MoveL 4578 to (-41.88, -24.72, -5.37) mm, rotated rx 180 ry 0 rz 90 deg; joints [72.599, -18.203, 86.885, 0, 21.318, 72.599]
  MoveL 4579 to (-43.16, -23.9, -5.78) mm, rotated rx -180 ry 0 rz 90 deg; joints [72.613, -18.208, 86.976, 0, 21.231, 72.613]
  MoveL 4580 to (-44.59, -23.38, -6.19) mm, rotated rx 180 ry 0 rz 90 deg; joints [72.616, -18.213, 87.072, 0, 21.141, 72.616]
  MoveL 4581 to (-46.1, -23.19, -6.59) mm, rotated rx -180 ry 0 rz 90 deg; joints [72.606, -18.218, 87.165, 0, 21.053, 72.606]
  MoveL 4582 to (-47.6, -23.37, -7) mm, rotated rx -180 ry 0 rz 90 deg; joints [72.585, -18.221, 87.251, 0, 20.97, 72.585]
  MoveL 4583 to (-71.99, -28.55, -7) mm, rotated rx 180 ry 0 rz 90 deg; joints [72.158, -18.582, 88.789, 0, 19.793, 72.158]
  MoveC 4584 to (-72.87, -28.82, -7) mm, rotated rx 180 ry 0 rz 90 deg; joints [72.139, -18.594, 88.842, 0, 19.752, 72.139] to (-73.69, -29.24, -7) mm, rotated rx 180 ry 0 rz 90 deg; joints [72.117, -18.605, 88.888, 0, 19.717, 72.117]
  MoveC 4585 to (-74.91, -30.54, -7) mm, rotated rx -180 ry 0 rz 90 deg; joints [72.06, -18.617, 88.942, 0, 19.676, 72.06] to (-75.35, -32.27, -7) mm, rotated rx 180 ry 0 rz 90 deg; joints [71.998, -18.615, 88.934, 0, 19.682, 71.998]
  MoveL 4586 to (-75.35, -70.6, -7) mm, rotated rx 180 ry 0 rz 90 deg; joints [70.733, -18.415, 88.068, 0, 20.347, 70.733]
  MoveL 4587 to (-75.33, -71.07, -7) mm, rotated rx 180 ry 0 rz 90 deg; joints [70.718, -18.412, 88.056, 0, 20.356, 70.718]
  MoveC 4588 to (-74.18, -73.67, -7) mm, rotated rx 180 ry 0 rz 90 deg; joints [70.646, -18.38, 87.918, 0, 20.462, 70.646] to (-71.55, -74.73, -7) mm, rotated rx -180 ry 0 rz 90 deg; joints [70.642, -18.332, 87.716, 0, 20.616, 70.642]
  MoveL 4589 to (-42.17, -74.5, -7) mm, rotated rx -180 ry 0 rz 90 deg; joints [70.98, -17.845, 85.724, 0, 22.121, 70.98]
  MoveL 4590 to (-35.54, -74.44, -7) mm, rotated rx -180 ry 0 rz 90 deg; joints [71.056, -17.73, 85.268, 0, 22.462, 71.056]
  MoveL 4591 to (-35.08, -74.42, -7) mm, rotated rx 180 ry 0 rz 90 deg; joints [71.061, -17.722, 85.237, 0, 22.486, 71.061]
  MoveC 4592 to (-32.87, -73.55, -7) mm, rotated rx 180 ry 0 rz 90 deg; joints [71.113, -17.689, 85.104, 0, 22.584, 71.113] to (-31.59, -71.55, -7) mm, rotated rx 180 ry 0 rz 90 deg; joints [71.192, -17.678, 85.063, 0, 22.615, 71.192]
  MoveL 4593 to (-31.32, -70.6, -7) mm, rotated rx -180 ry 0 rz 90 deg; joints [71.225, -17.679, 85.066, 0, 22.613, 71.225]
  MoveL 4594 to (-21.32, -32.17, -7) mm, rotated rx 180 ry 0 rz 90 deg; joints [72.567, -17.725, 85.245, 0, 22.479, 72.567]
  MoveL 4595 to (-18.98, -23.22, -7) mm, rotated rx 180 ry 0 rz 90 deg; joints [72.88, -17.732, 85.276, 0, 22.456, 72.88]
  MoveC 4596 to (-18.94, -21.18, -7) mm, rotated rx -180 ry 0 rz 90 deg; joints [72.946, -17.743, 85.317, 0, 22.426, 72.946] to (-19.96, -19.43, -7) mm, rotated rx 180 ry 0 rz 90 deg; joints [72.993, -17.77, 85.426, 0, 22.344, 72.993]
  MoveC 4597 to (-21.43, -18.37, -7) mm, rotated rx 180 ry 0 rz 90 deg; joints [73.013, -17.802, 85.551, 0, 22.251, 73.013] to (-23.22, -18.18, -7) mm, rotated rx 180 ry 0 rz 90 deg; joints [73.001, -17.834, 85.679, 0, 22.155, 73.001]
  MoveL 4598 to (-47.6, -23.37, -7) mm, rotated rx -180 ry 0 rz 90 deg; joints [72.585, -18.221, 87.251, 0, 20.97, 72.585]
  MoveL 4599 to (-46.03, -30.75, -7) mm, rotated rx 180 ry 0 rz 90 deg; joints [72.359, -18.156, 86.984, 0, 21.173, 72.359]
